		IF SIf.Par.bolEnableDoublePaperDetection THEN
			me.StateMachine.intStateNext := Base_PLC.cSTA_ERROR;
		END_IF
	ELSE	
		CASE me.SubStateMachine.intState OF
			// substate Wait paper - wait for the next paper if the buffer was empty
			// ------------------------------------------------------------------------
			PBC_CmdState.cSUB_WAITPAPER:
				IF NOT SIf.In.bolPaperAvailableExit.intern THEN
					IF SIf.In.bolCapacityReached.intern OR SIf.In.bolPaperAvailableEntry.intern THEN
						me.SubStateMachine.intStateNext := PBC_CmdState.cSUB_POSITIONSTARTbusy;
					END_IF
				ELSE
					me.SubStateMachine.intStateNext := cSUB_EVALUATEEJECT;
				END_IF
				
			// substate PositionStart busy
			// ------------------------------------------------------------------------
			PBC_CmdState.cSUB_POSITIONSTARTbusy:
				IF NOT SIf.In.bolPaperAvailableExit.intern THEN
					SIf.Cur.bolPaperBeforeEjectAvailable := SIf.In.bolCapacityReached.intern OR SIf.In.bolPaperAvailableEntry.intern;
					pDeStackerCIf^.Job.intACmd := BASE_PLC.cCMD_RUN;
					me.SubStateMachine.intStateNext := PBC_CmdState.cSUB_POSITIONbusy;
				ELSE
					me.SubStateMachine.intStateNext := cSUB_EVALUATEEJECT;
				END_IF
	
			// substate Position busy
			// ------------------------------------------------------------------------
			PBC_CmdState.cSUB_POSITIONbusy:
				IF me.SubStateMachine.udiTimeInState_ms <= SIf.Par.udiPaperTransportTime THEN
					IF SIf.In.bolPaperAvailableExit.intern THEN
						m_intRetry := 0;
						pDeStackerCIf^.Job.intACmd := BASE_PLC.cCMD_STOP;
						me.SubStateMachine.intStateNext := PBC_CmdState.cSUB_POSITIONSTOPbusy;
					END_IF
				ELSE
					IF SIf.Cur.bolPaperBeforeEjectAvailable OR SIf.In.bolCapacityReached.intern OR SIf.In.bolPaperAvailableEntry.intern THEN
						IF DINT_TO_UDINT(m_intRetry) < SIf.Par.udiPaperInjectRetries THEN
							pDeStackerCIf^.Job.intACmd := BASE_PLC.cCMD_STOP;
							m_intRetry := m_intRetry + 1;
							pfbAlarmCtrl^.setAlarm(CIf.Info.intCtrlId,INT_TO_UINT(E_ALM_PBC.PaperInjectRetry),m_intRetry,ADR(SIf.Alm),E_AlmState.RST,CIf.Job.eMe_ActivAlmClass);
							me.SubStateMachine.intStateNext := PBC_CmdState.cSUB_POSITIONRETRYSTOP;	
						ELSE
							m_intRetry := 0;
							pfbAlarmCtrl^.setAlarm(CIf.Info.intCtrlId,INT_TO_UINT(E_ALM_PBC.PaperInject),0,ADR(SIf.Alm),E_AlmState.RST,CIf.Job.eMe_ActivAlmClass);
							me.StateMachine.intStateNext := Base_PLC.cSTA_ERROR;	
						END_IF
					ELSE
						m_intRetry := 0;
						pDeStackerCIf^.Job.intACmd := BASE_PLC.cCMD_STOP;
						me.SubStateMachine.intStateNext := PBC_CmdState.cSUB_POSITIONSTOPbusy;
					END_IF 
				END_IF

				// Simulation
				IF CIf.SwCfg.bolSimulation THEN
					IF (me.SubStateMachine.udiTimeInState_ms > SIf.Par.udiSimPaperTransportTime) AND NOT SIf.In.bolPaperAvailableExit.intern THEN
						SIf.In.bolPaperAvailableExit.intern := TRUE;	
					END_IF
				END_IF
				// -----------------------------------
	
			// Wait that the moto stops
			// ------------------------------------------------------------------------
			PBC_CmdState.cSUB_POSITIONRETRYSTOP:
				IF pDeStackerCIf^.Job.intState = BASE_PLC.cSTA_STOP THEN
					me.SubStateMachine.intStateNext := PBC_CmdState.cSUB_POSITIONRETRYDELAY;
				END_IF

			// Stop the motor and way for x ms
			// ------------------------------------------------------------------------
			PBC_CmdState.cSUB_POSITIONRETRYDELAY:
				IF me.SubStateMachine.udiTimeInState_ms > SIf.Par.udiPaperInjectRetryPauseTime_ms THEN
					me.SubStateMachine.intStateNext := PBC_CmdState.cSUB_POSITIONSTARTbusy;
				END_IF

			// substate PositionStop busy
			// ------------------------------------------------------------------------
			PBC_CmdState.cSUB_POSITIONSTOPbusy:
				IF pDeStackerCIf^.Job.intState = BASE_PLC.cSTA_STOP THEN
					me.SubStateMachine.intStateNext := PBC_CmdState.cSUB_EVALUATEEJECT;
				END_IF

			// substate Evaluate Eject
			// ------------------------------------------------------------------------
			PBC_CmdState.cSUB_EVALUATEEJECT:
				bolSaberStopDestack		:= SIf.Par.bolStopReleaseItems AND SIf.Cfg.bolEnableSaberStopDeStack;

				// Eject next paper if there are still paper to edject or endless ejection
				IF (((SIf.Cur.uinPaperToEjectCount > 0) AND NOT SIf.Par.bolAutomaticMode AND NOT bolSaberStopDestack) 
					OR (SIf.Par.bolAutomaticMode AND NOT bolSaberStopDestack)) THEN 
					// Make a delay from sheet to sheet if it is not the first sheet
					IF SIf.In.bolPaperAvailableExit.intern THEN
						IF   (SIf.Cur.uinSheetToSheetTime > SIf.Par.udiSheetToSheetTime) 
						  OR ((SIf.Cur.uinPaperToEjectCount = SIf.Cur.uinPaperToEjectParameter) AND NOT SIf.Par.bolAutomaticMode) THEN
							SIf.Cur.uinSheetToSheetTime := 0;
							me.SubStateMachine.intStateNext := PBC_CmdState.cSUB_EJECTSTARTbusy;
						END_IF
					ELSE
						me.SubStateMachine.intStateNext := PBC_CmdState.cSUB_WAITPAPER;
					END_IF
				ELSE
					me.StateMachine.intStateNext := cSTA_STOPBusy;
				END_IF
	
			// substate EjectStart busy
			// ------------------------------------------------------------------------
			PBC_CmdState.cSUB_EJECTSTARTbusy:
				pDeStackerCIf^.Job.intACmd := BASE_PLC.cCMD_RUN;
				SIf.Cur.uinPaperToPaperTime_ms := UDINT_TO_UINT((m_uinPaperHight_mm + 100) * 1000 / p_fbDeStacker^.CtrlSIf^.Par.rBeltParam.uinBeltSpeed);
				SIf.Par.udiSimPaperToPaperTransportTime := SIf.Cur.uinPaperToPaperTime_ms / 3; 
				me.SubStateMachine.intStateNext := PBC_CmdState.cSUB_EJECTbusy;
	
			// substate Eject busy
			// ------------------------------------------------------------------------
			PBC_CmdState.cSUB_EJECTbusy:
				IF NOT SIf.In.bolPaperAvailableExit.intern AND NOT SIf.Cfg.bolUseTurnTableSensorForEject THEN
					pDeStackerCIf^.Job.intACmd := BASE_PLC.cCMD_STOP;
					me.SubStateMachine.intStateNext := PBC_CmdState.cSUB_EJECTSTOPbusy;
				END_IF
	
				IF SIf.In.bolTurnTableMiddleSensor.intern AND SIf.Cfg.bolUseTurnTableSensorForEject THEN
					pDeStackerCIf^.Job.intACmd := BASE_PLC.cCMD_STOP;
					me.SubStateMachine.intStateNext := PBC_CmdState.cSUB_WAITPAPERGONETABLE;
				END_IF
				
				IF (me.SubStateMachine.udiTimeInState_ms > SIf.Cur.uinPaperToPaperTime_ms) THEN
					pfbAlarmCtrl^.setAlarm(CIf.Info.intCtrlId,INT_TO_UINT(E_ALM_PBC.PaperTransport),0,ADR(SIf.Alm),E_AlmState.RST,CIf.Job.eMe_ActivAlmClass);
					me.StateMachine.intStateNext := Base_PLC.cSTA_ERROR;	
				END_IF

				// Simulation
				IF CIf.SwCfg.bolSimulation THEN
					IF (me.SubStateMachine.udiTimeInState_ms > SIf.Par.udiSimPaperToPaperTransportTime) THEN
						IF SIf.Cfg.bolUseTurnTableSensorForEject THEN
							SIf.In.bolTurnTableMiddleSensor.intern := TRUE;
						ELSE
							SIf.In.bolPaperAvailableExit.intern := FALSE;	
						END_IF	
					END_IF
				END_IF
				// -----------------------------------
	
			// substate Wait Paper Gone Table - Wait until the paper is gone from the turn table
			// ------------------------------------------------------------------------
			PBC_CmdState.cSUB_WAITPAPERGONETABLE:
				IF NOT SIf.In.bolTurnTableMiddleSensor.intern THEN
					me.SubStateMachine.intStateNext := PBC_CmdState.cSUB_EJECTSTOPbusy;
				END_IF

				// Simulation
				IF CIf.SwCfg.bolSimulation THEN
					IF (me.SubStateMachine.udiTimeInState_ms > SIf.Par.udiSimPaperToPaperTransportTime) THEN
						SIf.In.bolTurnTableMiddleSensor.intern := FALSE;
					END_IF
				END_IF
				// -----------------------------------

	
			// substate EjectStop busy
			// ------------------------------------------------------------------------
			PBC_CmdState.cSUB_EJECTSTOPbusy:
				IF pDeStackerCIf^.Job.intState = BASE_PLC.cSTA_STOP THEN
					IF SIf.Cur.uinPaperToEjectCount > 0 THEN
						SIf.Cur.uinPaperToEjectCount := SIf.Cur.uinPaperToEjectCount - 1;
					END_IF
	
					me.SubStateMachine.intStateNext := PBC_CmdState.cSUB_POSITIONSTARTbusy;
				END_IF
		END_CASE
	END_IF
	
	CASE me.SubStateMachine.intState OF
		PBC_CmdState.cSUB_WAITPAPER,
		PBC_CmdState.cSUB_EVALUATEEJECT:
			IF (me.intCmd = BASE_PLC.cCMD_STOP) THEN 
					me.StateMachine.intStateNext := BASE_PLC.cSTA_STOPBusy;
			END_IF
	END_CASE
	
	SIf.Cur.uinSheetToSheetTime := UDINT_TO_UINT(SIf.Cur.uinSheetToSheetTime + me.FUBInfo.udiSample_ms);
END_IF


//--------------------------------------------------------------------------------------
// Exit action
IF (me.StateMachine.intState<>me.StateMachine.intStateNext) THEN
	me.SubStateMachine.intState 	:= BASE_PLC.cSTA_INITIALIZED;
	me.SubStateMachine.intStateNext := BASE_PLC.cSTA_INITIALIZED;
END_IF
END_METHOD

{attribute 'object_name' := 'sta_RUNbusy'}
METHOD PROTECTED sta_RUNbusy : BOOL
// state implemetation
//--------------------------------------------------------------------------------------
// Entry action
IF (me.StateMachine.intState<>me.StateMachine.intStateLastCycle) THEN
	me.StateMachine.intStateLastCycle := me.StateMachine.intState;

	IF (CIf.SwCfg.bolSimulation) THEN
		SIf.In.bolCapacityReached.intern := FALSE;
		SIf.In.bolPaperAvailableEntry.intern := TRUE;
		SIf.In.bolPaperAvailableExit.intern := TRUE;
	END_IF

	SIf.Out.bolAirOn.intern := TRUE;
	
	pDeStackerCIf^.Job.intACmd := BASE_PLC.cCMD_STOP;
	pBeltCIf^.Job.intACmd := BASE_PLC.cCMD_RUN;
	
	// clear alarm
	pfbAlarmCtrl^.setAlarm(CIf.Info.intCtrlId,INT_TO_UINT(E_ALM_PBC.DoNotReleaseItems),0,ADR(SIf.Alm),E_AlmState.CLR,CIf.Job.eMe_ActivAlmClass);
END_IF


//--------------------------------------------------------------------------------------
// Cyclic action
IF (me.StateMachine.intState=me.StateMachine.intStateLastCycle) THEN
	IF SIf.Par.bolAutomaticMode THEN
		SIf.Cur.uinPaperToEjectParameter := 0;
		SIf.Cur.uinPaperToEjectCount := 0;
		me.StateMachine.intStateNext := BASE_PLC.cSTA_RUN;
	ELSE	
		IF me.intCmd = PBC_CmdState.cCMD_SINGLE THEN
			SIf.Cur.uinPaperToEjectParameter := 1;
			SIf.Cur.uinPaperToEjectCount := 1;
	
			IF NOT SIf.In.bolPaperAvailableExit.intern AND NOT SIf.In.bolPaperAvailableEntry.intern THEN
				pfbAlarmCtrl^.setAlarm(CIf.Info.intCtrlId,INT_TO_UINT(E_ALM_PBC.BufferEmpty),0,ADR(SIf.Alm),E_AlmState.RST,CIf.Job.eMe_ActivAlmClass);
			END_IF
	
			me.StateMachine.intStateNext := BASE_PLC.cSTA_RUN;
		ELSE
			IF me.StateMachine.intStateHistory = Base_PLC.cSTA_OFF THEN
				CIf.Job.intACmd := cCMD_DONE;
				CIf.Job.intMCmd := cCMD_DONE;
				me.StateMachine.intStateNext := BASE_PLC.cSTA_STOPBusy;
			ELSE
				SIf.Cur.uinPaperToEjectParameter := UDINT_TO_UINT(SIf.Par.udiSheetToEject);
				SIf.Cur.uinPaperToEjectCount := UDINT_TO_UINT(SIf.Par.udiSheetToEject);
		
				IF SIf.Par.udiSheetToEject > 0 THEN
					me.StateMachine.intStateNext := BASE_PLC.cSTA_RUN;
				ELSE
					CIf.Job.intACmd := cCMD_DONE;
					CIf.Job.intMCmd := cCMD_DONE;
					me.StateMachine.intStateNext := BASE_PLC.cSTA_STOPBusy;
				END_IF
			END_IF
		END_IF
	END_IF
END_IF


//--------------------------------------------------------------------------------------
// Exit action
IF (me.StateMachine.intState<>me.StateMachine.intStateNext) THEN
	;
END_IF
END_METHOD

{attribute 'object_name' := 'sta_STOP'}
METHOD PROTECTED sta_STOP : BOOL
// state implemetation
//--------------------------------------------------------------------------------------
// Entry action
IF (me.StateMachine.intState<>me.StateMachine.intStateLastCycle) THEN
	me.StateMachine.intStateLastCycle := me.StateMachine.intState;

	IF CIf.SwCfg.bolSimulation THEN
		SIf.In.bolPaperAvailableEntry.intern := TRUE;
		SIf.In.bolDoublePaperDetection.intern := FALSE;	
		SIf.In.bolPaperAvailableExit.intern := FALSE;	
		SIf.In.bolCapacityReached.intern := TRUE;
	END_IF
	
	IF me.intCmd = Base_PLC.cCMD_RUN THEN
		CIf.Job.intACmd := Base_PLC.cCMD_DONE;
		CIf.Job.intMCmd := Base_PLC.cCMD_DONE;
	END_IF
	
	me.SubStateMachine.intState 	:= PBC_CmdState.cSUB_POSITIONSTARTbusy;
	me.SubStateMachine.intStateNext := PBC_CmdState.cSUB_POSITIONSTARTbusy;
END_IF

//--------------------------------------------------------------------------------------
// Cyclic action
IF (me.StateMachine.intState=me.StateMachine.intStateLastCycle) THEN
	CASE me.SubStateMachine.intState OF
		// substate Wait paper - wait for the next paper if the buffer was empty
		// ------------------------------------------------------------------------
		PBC_CmdState.cSUB_WAITPAPER:
			IF SIf.In.bolPaperAvailableExit.intern THEN
				me.SubStateMachine.intStateNext := PBC_CmdState.cSUB_READYEJECT;
			ELSE
				IF SIf.In.bolCapacityReached.intern OR SIf.In.bolPaperAvailableEntry.intern THEN
					me.SubStateMachine.intStateNext := PBC_CmdState.cSUB_POSITIONSTARTbusy;
				END_IF
			END_IF
			
		// substate Wait paper - wait for the next paper if the buffer was empty
		// ------------------------------------------------------------------------
		PBC_CmdState.cSUB_POSITIONSTARTbusy:
			IF NOT SIf.In.bolPaperAvailableExit.intern THEN
				SIf.Cur.bolPaperBeforeEjectAvailable := SIf.In.bolCapacityReached.intern OR SIf.In.bolPaperAvailableEntry.intern;
				pDeStackerCIf^.Job.intACmd := BASE_PLC.cCMD_RUN;
				me.SubStateMachine.intStateNext := PBC_CmdState.cSUB_POSITIONbusy;
			ELSE
				me.SubStateMachine.intStateNext := cSUB_READYEJECT;
			END_IF

		// substate Wait paper - wait for the next paper if the buffer was empty
		// ------------------------------------------------------------------------
		PBC_CmdState.cSUB_POSITIONbusy:
			IF me.SubStateMachine.udiTimeInState_ms > SIf.Par.udiPaperTransportTime THEN
				IF SIf.Cur.bolPaperBeforeEjectAvailable OR SIf.In.bolCapacityReached.intern OR SIf.In.bolPaperAvailableEntry.intern THEN
					pfbAlarmCtrl^.setAlarm(CIf.Info.intCtrlId,INT_TO_UINT(E_ALM_PBC.PaperTransport),0,ADR(SIf.Alm),E_AlmState.RST,CIf.Job.eMe_ActivAlmClass);
					me.StateMachine.intStateNext := Base_PLC.cSTA_ERROR;	
				ELSE
					pDeStackerCIf^.Job.intACmd := BASE_PLC.cCMD_STOP;
					me.SubStateMachine.intStateNext := PBC_CmdState.cSUB_POSITIONSTOPbusy;
				END_IF 
			ELSE
				IF SIf.In.bolPaperAvailableExit.intern THEN
					pDeStackerCIf^.Job.intACmd := BASE_PLC.cCMD_STOP;
					me.SubStateMachine.intStateNext := PBC_CmdState.cSUB_POSITIONSTOPbusy;
				END_IF
			END_IF
			
			// Simulation
			IF CIf.SwCfg.bolSimulation THEN
				IF (me.SubStateMachine.udiTimeInState_ms > SIf.Par.udiSimPaperTransportTime) AND NOT SIf.In.bolPaperAvailableExit.intern THEN
					SIf.In.bolPaperAvailableExit.intern := TRUE;	
				END_IF
			END_IF
			// -----------------------------------

		// substate Wait paper - wait for the next paper if the buffer was empty
		// ------------------------------------------------------------------------
		PBC_CmdState.cSUB_POSITIONSTOPbusy:
			IF pDeStackerCIf^.Job.intState = BASE_PLC.cSTA_STOP THEN
				IF SIf.In.bolPaperAvailableExit.intern THEN
					me.SubStateMachine.intStateNext := PBC_CmdState.cSUB_READYEJECT;
				ELSE
					me.SubStateMachine.intStateNext := PBC_CmdState.cSUB_WAITPAPER;
				END_IF
			END_IF
		PBC_CmdState.cSUB_READYEJECT:
			IF NOT SIf.In.bolPaperAvailableExit.intern THEN
				me.SubStateMachine.intStateNext := PBC_CmdState.cSUB_WAITPAPER;
			END_IF
	END_CASE

	CASE me.SubStateMachine.intState OF
		PBC_CmdState.cSUB_WAITPAPER,
		PBC_CmdState.cSUB_READYEJECT:
			IF me.intCmd = PBC_CmdState.cCMD_SINGLE THEN
				me.StateMachine.intStateNext := BASE_PLC.cSTA_RUNBusy;
			END_IF
		
			IF ((me.intCmd = BASE_PLC.cCMD_RUN) AND (NOT SIf.Par.bolStopReleaseItems AND SIf.Cfg.bolEnableSaberStopDeStack))
				OR ((me.intCmd = BASE_PLC.cCMD_RUN) AND NOT SIf.Cfg.bolEnableSaberStopDeStack) THEN
				me.StateMachine.intStateNext := BASE_PLC.cSTA_RUNBusy;
			END_IF

			IF (SIf.Par.bolAutomaticMode AND (NOT SIf.Par.bolStopReleaseItems AND SIf.Cfg.bolEnableSaberStopDeStack))
				OR (SIf.Par.bolAutomaticMode AND NOT SIf.Cfg.bolEnableSaberStopDeStack) THEN
				me.StateMachine.intStateNext := BASE_PLC.cSTA_RUNBusy;
			END_IF
	END_CASE
END_IF


//--------------------------------------------------------------------------------------
// Exit action
IF (me.StateMachine.intState<>me.StateMachine.intStateNext) THEN
	me.SubStateMachine.intState 	:= BASE_PLC.cSTA_INITIALIZED;
	me.SubStateMachine.intStateNext := BASE_PLC.cSTA_INITIALIZED;
END_IF
END_METHOD

{attribute 'object_name' := 'sta_STOPbusy'}
METHOD PROTECTED sta_STOPbusy : BOOL
// state implemetation
//--------------------------------------------------------------------------------------
// Entry action
IF (me.StateMachine.intState<>me.StateMachine.intStateLastCycle) THEN
	me.StateMachine.intStateLastCycle := me.StateMachine.intState;

	pDeStackerCIf^.Job.intACmd := BASE_PLC.cCMD_STOP;
	
	// set alarm
	pfbAlarmCtrl^.setAlarm(CIf.Info.intCtrlId,INT_TO_UINT(E_ALM_PBC.DoNotReleaseItems),0,ADR(SIf.Alm),E_AlmState.SET,CIf.Job.eMe_ActivAlmClass);
END_IF


//--------------------------------------------------------------------------------------
// Cyclic action
IF (me.StateMachine.intState=me.StateMachine.intStateLastCycle) THEN
	me.StateMachine.intStateNext := BASE_PLC.cSTA_STOP;
END_IF


//--------------------------------------------------------------------------------------
// Exit action
IF (me.StateMachine.intState<>me.StateMachine.intStateNext) THEN
	;
END_IF
END_METHOD

{attribute 'object_name' := 'StateMachine'}
METHOD PROTECTED StateMachine : BOOL
SUPER^.StateMachine();

// main statemachine of base controller
CASE me.StateMachine.intState OF
	BASE_PLC.cSTA_RUN:
		THIS^.sta_RUN();
	BASE_PLC.cSTA_RUNBusy:
		THIS^.sta_RUNbusy();
    BASE_PLC.cSTA_STOPBusy: 
        THIS^.sta_STOPbusy();
    BASE_PLC.cSTA_STOP: 
        THIS^.sta_STOP();
	PBC_CmdState.cSTA_INITbusy:
		THIS^.sta_INITbusy();
END_CASE;
END_METHOD

END_FUNCTION_BLOCK

// POUs/Controller/Lvl2/PCE [Paper Belt Corner Element]/helper/cycle_Pce
FUNCTION cycle_Pce : BOOL
VAR_INPUT
	pPce: POINTER TO T_PCE;
END_VAR

pPce^.ctrl.fbPce_PtbIn_Umc.In_bolEmoOk				:= pPce^.io.In_bolUmcIn_EmoOk;
pPce^.ctrl.fbPce_PtbIn_Umc.In_uinStatus				:= pPce^.io.In_uinUmcIn_Status;
pPce^.ctrl.fbPce_PtbIn_Umc.In_intMotorActualSpeed	:= pPce^.io.In_uinUmcIn_ActualSpeed;
pPce^.ctrl.fbPce_PtbIn_Umc.In_uinMotorSetSpeed		:= pPce^.io.In_uinUmcIn_SetSpeed;
pPce^.ctrl.fbPce_PtbIn_Umc.In_uinECATState			:= pPce^.io.In_uinUmcIn_ECatState;
pPce^.ctrl.fbPce_PtbIn_Umc.In_strNetId				:= pPce^.io.In_strUmcIn_ECatNetId;
pPce^.ctrl.fbPce_PtbIn_Umc.In_uintPort				:= pPce^.io.In_uinUmcIn_ECatPort;
pPce^.ctrl.fbPce_PtbIn_Umc();
pPce^.io.Out_uinUmcIn_SetSpeed						:= pPce^.ctrl.fbPce_PtbIn_Umc.Out_uinSpeedSetpoint;
pPce^.io.Out_uinUmcIn_Control						:= pPce^.ctrl.fbPce_PtbIn_Umc.Out_uinControl;

pPce^.ctrl.fbPce_PtbIn_Vpc.In_bolPumpOk				:= pPce^.io.In_bolVpc_PumpOk;
pPce^.ctrl.fbPce_PtbIn_Vpc.In_bolVacuumOk			:= pPce^.io.In_bolVpc_VacuumSensor;
pPce^.ctrl.fbPce_PtbIn_Vpc();
pPce^.io.Out_bolVpc_PumpOn							:= pPce^.ctrl.fbPce_PtbIn_Vpc.Out_bolVaccumPumpOn;

pPce^.ctrl.fbPce_PtbIn.In_bolBeltEntrySensor		:= pPce^.io.In_bolInputSensor;
pPce^.ctrl.fbPce_PtbIn.In_bolBeltExitSensor			:= pPce^.io.In_bolCornerSensor;
pPce^.ctrl.fbPce_PtbIn();

pPce^.ctrl.fbPce_PtbOut_Umc.In_bolEmoOk				:= pPce^.io.In_bolUmcIn_EmoOk;
pPce^.ctrl.fbPce_PtbOut_Umc.In_uinStatus			:= pPce^.io.In_uinUmcOut_Status;
pPce^.ctrl.fbPce_PtbOut_Umc.In_intMotorActualSpeed	:= pPce^.io.In_uinUmcOut_ActualSpeed;
pPce^.ctrl.fbPce_PtbOut_Umc.In_uinMotorSetSpeed		:= pPce^.io.In_uinUmcOut_SetSpeed;
pPce^.ctrl.fbPce_PtbOut_Umc.In_uinECATState			:= pPce^.io.In_uinUmcOut_ECatState;
pPce^.ctrl.fbPce_PtbOut_Umc.In_strNetId				:= pPce^.io.In_strUmcOut_ECatNetId;
pPce^.ctrl.fbPce_PtbOut_Umc.In_uintPort				:= pPce^.io.In_uinUmcOut_ECatPort;
pPce^.ctrl.fbPce_PtbOut_Umc();
pPce^.io.Out_uinUmcOut_SetSpeed						:= pPce^.ctrl.fbPce_PtbOut_Umc.Out_uinSpeedSetpoint;
pPce^.io.Out_uinUmcOut_Control						:= pPce^.ctrl.fbPce_PtbOut_Umc.Out_uinControl;

pPce^.ctrl.fbPce_PtbOut.In_bolBeltEntrySensor		:= pPce^.io.In_bolCornerSensor;
pPce^.ctrl.fbPce_PtbOut.In_bolBeltExitSensor		:= pPce^.io.In_bolOutputSensor;
pPce^.ctrl.fbPce_PtbOut();

pPce^.ctrl.fbPce.In_bolPaperAvailable				:=pPce^.io.In_bolCornerSensor;
pPce^.ctrl.fbPce();
pPce^.io.Out_bolVacuumValveIn						:= pPce^.ctrl.fbPce.Out_bolVacuumValveIn;
pPce^.io.Out_bolVacuumValveOut						:= pPce^.ctrl.fbPce.Out_bolVacuumValveOut;

END_FUNCTION

// POUs/Controller/Lvl2/PCE [Paper Belt Corner Element]/helper/init_Pce
FUNCTION init_Pce : BOOL
VAR_INPUT
	pPce			: POINTER TO T_PCE;
	/// instance array of all controller instances
	pCtrlInst		: POINTER TO fb_CtrlBase;
	/// common interface array of all controllers (main use for PLC)
	pCtrlCIf		: POINTER TO T_Ctrl_CIf;
END_VAR

pPce^.ctrl.fbPce_PtbIn_Vpc.iniAllCtrlArrays(pCtrlInst,pCtrlCIf,pPce^.id.Pce_PtbIn_Vpc);
pPce^.ctrl.fbPce_PtbIn_Umc.iniAllCtrlArrays(pCtrlInst,pCtrlCIf,pPce^.id.Pce_PtbIn_Umc);
pPce^.ctrl.fbPce_PtbIn.iniAllCtrlArrays(pCtrlInst,pCtrlCIf,pPce^.id.Pce_PtbIn);
pPce^.ctrl.fbPce_PtbIn.Drive := ADR(pPce^.ctrl.fbPce_PtbIn_Umc);
pPce^.ctrl.fbPce_PtbIn.VacuumPump := ADR(pPce^.ctrl.fbPce_PtbIn_Vpc);

pPce^.ctrl.fbPce_PtbOut_Umc.iniAllCtrlArrays(pCtrlInst,pCtrlCIf,pPce^.id.Pce_PtbOut_Umc);
pPce^.ctrl.fbPce_PtbOut.iniAllCtrlArrays(pCtrlInst,pCtrlCIf,pPce^.id.Pce_PtbOut);
pPce^.ctrl.fbPce_PtbOut.Drive := ADR(pPce^.ctrl.fbPce_PtbOut_Umc);

pPce^.ctrl.fbPce.iniAllCtrlArrays(pCtrlInst,pCtrlCIf,pPce^.id.Pce);
pPce^.ctrl.fbPce.DriveIn := ADR(pPce^.ctrl.fbPce_PtbIn);
pPce^.ctrl.fbPce.DriveOut := ADR(pPce^.ctrl.fbPce_PtbOut);

END_FUNCTION

// POUs/Controller/Lvl2/PCE [Paper Belt Corner Element]/FB_PCE
FUNCTION_BLOCK FB_PCE EXTENDS FB_CtrlBase
VAR_INPUT
	In_bolPaperAvailable: BOOL;
END_VAR
VAR_OUTPUT
	Out_bolVacuumValveIn: BOOL;
	Out_bolVacuumValveOut: BOOL;
END_VAR
VAR
	/// Specific interface struct for public access
	SIf: T_Ctrl_SIf_PCE;
	///pointer to function block
	p_fbMotorIn: POINTER TO FB_PTB;
	pMotorInCIf: POINTER TO T_Ctrl_CIf;
	p_fbMotorOut: POINTER TO FB_PTB;
	pMotorOutCIf: POINTER TO T_Ctrl_CIf;
END_VAR

(*__________________________________________________________________________________________________
¦	
¦	Vistaprint Schweiz GmbH
¦	CH - 8401 Winterthur
¦
¦	www.vistaprint.ch - info@vistaprint.ch
¦___________________________________________________________________________________________________

Function desription:
Vacuum Pump implementation. 


History:
Version		Date			Author		Comment
---------------------------------------------------------------------------------------------------
0.00.1		09.07.2013		PC			Start history
___________________________________________________________________________________________________*)


SUPER^();

{attribute 'object_name' := 'Always'}
METHOD PROTECTED Always : BOOL
SUPER^.Always();

// ----------------------------------------------------------------------------------
// cyclic actions outside of statemachine
IF (me.StateMachine.intState<>cSTA_SINGLE_ANSWER) THEN
	
	; // always error supervision
	
END_IF

// ----------------------------------------------------------------------------------
// Conditions Always
IF (((me.Alarm.eActivAlmClass=E_AlmClass.EOFF) OR (me.Alarm.eActivAlmClass=E_AlmClass.OFF) OR (me.intCmd=cCMD_OFF) OR (me.intCmd=BASE_PLC.cCMD_EOFF))
		 AND (me.StateMachine.intState<>cSTA_ERROR) AND (me.StateMachine.intState<>cSTA_ERRORQuit) AND
		(me.StateMachine.intState<>cSTA_OFF) AND (me.StateMachine.intState<>cSTA_OFFBusy)) THEN
	// alarm evt EOFF, OFF or cmd off
	me.StateMachine.intStateNext := cSTA_OFFBusy;
END_IF
END_METHOD

{attribute 'object_name' := 'CtrlInit'}
METHOD CtrlInit : BOOL
SUPER^.CtrlInit();

pMotorInCIf := p_fbMotorIn^.CtrlCIf;
pMotorOutCIf := p_fbMotorOut^.CtrlCIf;

AddChild(p_fbMotorIn^);
AddChild(p_fbMotorOut^);
END_METHOD

PROPERTY PUBLIC CtrlSIf : POINTER TO T_Ctrl_SIf_PCE
GET
CtrlSIf := ADR(SIf);
END_GET
END_PROPERTY

PROPERTY DriveIn : POINTER TO FB_PTB
GET
DriveIn := p_fbMotorIn;
END_GET
SET
p_fbMotorIn := DriveIn;
END_SET
END_PROPERTY

PROPERTY DriveOut : POINTER TO FB_PTB
GET
DriveOut := p_fbMotorOut;
END_GET
SET
p_fbMotorOut := DriveOut;
END_SET
END_PROPERTY

{attribute 'object_name' := 'FB_init'}
METHOD FB_init : BOOL
VAR_INPUT
	/// if TRUE, the retain variables are initialized (warm start / cold start)
	bInitRetains: BOOL;
	/// if TRUE, the instance afterwards gets moved into the copy code (online change)
	bInCopyCode: BOOL;
END_VAR
VAR
	iIdx: UINT;
	iLength: UINT;
END_VAR
//------------------------------------------------------------------------------------------------------------------------
// to manually change in new FUB implementation!!!
// define valid commands for this controller
iLength := SIZEOF(CIf.Job.aCmdList)/SIZEOF(CIf.Job.aCmdList[0]);
iIdx := 0;

WHILE (iIdx < iLength) AND (CIf.Job.aCmdList[iIdx].intCmd <> cCMD_INITIALIZED) DO
	iIdx := iIdx + 1; 
END_WHILE

IF (iIdx < iLength) THEN
// Add configuration of own comands	
	CIf.Job.aCmdList[iIdx].intCmd := BASE_PLC.cCMD_RUN;
	CIf.Job.aCmdList[iIdx].strName := 'Run'; 
	CIf.Job.aCmdList[iIdx].bolAvailable := TRUE;
	iIdx := iIdx + 1;
	CIf.Job.aCmdList[iIdx].intCmd := BASE_PLC.cCMD_STOP;
	CIf.Job.aCmdList[iIdx].strName := 'Stop'; 
	CIf.Job.aCmdList[iIdx].bolAvailable := TRUE;
ELSE
	// Error if the aCmdList Array is to small
END_IF

// set name of class/typ
CIf.Info.strType := 'FB_PCE';
CIf.Info.strFullName := 'Paper Corner Element';

// set alarm class

SIf.Alm[E_ALM_PCE.PaperSensorError].eAlmClass := Base_PLC.E_AlmClass.TSTOP;
SIf.Alm[E_ALM_PCE.PaperSensorError].strText := 'Paper detected to long' ;


//*******************************************************************************
// initial values
//*******************************************************************************

// software configuration
CIf.SwCfg.bolExist := TRUE;
CIf.SwCfg.bolEnable := TRUE;
CIf.SwCfg.bolSimulation := FALSE;

// parameter
SIf.Par.uinPaperExitTime_ms			:= 3000;
SIf.Par.uinSimPaperExitTime_ms		:= SIf.Par.uinPaperExitTime_ms / 2;
SIf.Par.uinPaperEntryDelayTime_ms   := 220;
END_METHOD

{attribute 'object_name' := 'getCmdState'}
METHOD PROTECTED getCmdState : STRING
VAR_INPUT
	intCmdState: INT;
	bolState: BOOL;
END_VAR
getCmdState := SUPER^.getCmdState(intCmdState:=intCmdState,bolState:=bolState); // get global/base defined cmds/states
END_METHOD

{attribute 'object_name' := 'getCtrlSIf'}
METHOD getCtrlSIf : POINTER TO T_Ctrl_SIf_PCE
getCtrlSIf := ADR(SIf);
END_METHOD

{attribute 'object_name' := 'IoInBridge'}
METHOD PROTECTED IoInBridge : BOOL
// digitale and analoge inputs read from hardware or forcing
SIf.In.bolPaperAvailable.map := THIS^.In_bolPaperAvailable;

IF (CIf.SwCfg.bolSimulation = FALSE) THEN
	getInBol(CIf.Job.bolIoForce,ADR(SIf.In.bolPaperAvailable));
ELSE
	;//simulation of global IO
END_IF
END_METHOD

{attribute 'object_name' := 'IoOutBridge'}
METHOD PROTECTED IoOutBridge : BOOL
VAR
	bolSwitchValvesOff: BOOL;
END_VAR
// digitale and analoge inputs read from hardware or forcing
IF (CIf.SwCfg.bolSimulation = FALSE) THEN
	setOutBol(CIf.Job.bolIoForce ,ADR(SIf.Out.bolVacuumValveIn));
	setOutBol(CIf.Job.bolIoForce ,ADR(SIf.Out.bolVacuumValveOut));

	THIS^.Out_bolVacuumValveIn := SIf.Out.bolVacuumValveIn.map;
	THIS^.Out_bolVacuumValveOut := SIf.Out.bolVacuumValveOut.map;
END_IF
END_METHOD

ACTION PaperExitValveActive:
SIf.Out.bolVacuumValveIn.intern := FALSE;
SIf.Out.bolVacuumValveOut.intern := TRUE;
END_ACTION

ACTION PaperInputValveActive:
SIf.Out.bolVacuumValveIn.intern := TRUE;
SIf.Out.bolVacuumValveOut.intern := FALSE;
END_ACTION

{attribute 'object_name' := 'sta_ERROR'}
METHOD PROTECTED sta_ERROR : BOOL
// state implemetation
//--------------------------------------------------------------------------------------
// Entry action
	IF (me.StateMachine.intState<>me.StateMachine.intStateLastCycle) THEN
		me.StateMachine.intStateHistory := me.StateMachine.intStateLastCycle; // -> possibillity to go back to state before error
		me.StateMachine.intStateLastCycle := me.StateMachine.intState;
		p_fbMotorIn^.CtrlCIf^.Job.intACmd := BASE_PLC.cCMD_STOP;
		p_fbMotorOut^.CtrlCIf^.Job.intACmd := BASE_PLC.cCMD_STOP;
	END_IF


//--------------------------------------------------------------------------------------
// Cyclic action
	IF (me.StateMachine.intState=me.StateMachine.intStateLastCycle) THEN
		
		;
		
		
		// State Change Condition
		IF (CIf.Job.bolAlmReset = TRUE) THEN
			me.StateMachine.intStateNext := cSTA_ERRORQuit;
		END_IF
	END_IF




//--------------------------------------------------------------------------------------
// Exit action
	IF (me.StateMachine.intState<>me.StateMachine.intStateNext) THEN
		;
	END_IF
END_METHOD

{attribute 'object_name' := 'sta_ERRORQuit'}
METHOD PROTECTED sta_ERRORQuit : BOOL
// state implemetation
//--------------------------------------------------------------------------------------
// Entry action
	IF (me.StateMachine.intState<>me.StateMachine.intStateLastCycle) THEN
		me.StateMachine.intStateLastCycle := me.StateMachine.intState;
		
	END_IF


//--------------------------------------------------------------------------------------
// Cyclic action
	IF (me.StateMachine.intState=me.StateMachine.intStateLastCycle) THEN
		
		;
		// evtl. wait time if reset of device is necessary and then decide to go to states or ERROR state
		IF (CIf.Job.bolAlmReset = TRUE) THEN
			CIf.Job.eMe_ActivAlmClass := E_AlmClass.NONE; // reset feedback channel for parent
			CIf.Job.bolAlmReset := FALSE;
		END_IF
		
		// State Change Condition
		IF (CIf.Job.bolAlmReset = FALSE) THEN
			IF (me.StateMachine.intStateHistory<=BASE_PLC.cSTA_PON) THEN
				me.StateMachine.intStateNext := BASE_PLC.cSTA_PONBusy;
			END_IF;

			CASE me.intCmd OF
				BASE_PLC.cCMD_OFF:
					me.StateMachine.intStateNext := BASE_PLC.cSTA_OFFBusy;
				BASE_PLC.cCMD_RUN:
					me.StateMachine.intStateNext := BASE_PLC.cSTA_RUNBusy;
			ELSE
				CASE me.StateMachine.intStateHistory OF
					BASE_PLC.cSTA_RUN:
						me.StateMachine.intStateNext := BASE_PLC.cSTA_RUNBusy;
					BASE_PLC.cSTA_OFF:
						me.StateMachine.intStateNext := BASE_PLC.cSTA_OFFBusy;
					BASE_PLC.cSTA_STOP:
						me.StateMachine.intStateNext := BASE_PLC.cSTA_STOPBusy;
				END_CASE
			END_CASE
		END_IF
	END_IF




//--------------------------------------------------------------------------------------
// Exit action
	IF (me.StateMachine.intState<>me.StateMachine.intStateNext) THEN
		;
	END_IF
END_METHOD

{attribute 'object_name' := 'sta_OFF'}
METHOD PROTECTED sta_OFF : BOOL
// state implemetation
//--------------------------------------------------------------------------------------
// Entry action
	IF (me.StateMachine.intState<>me.StateMachine.intStateLastCycle) THEN
		me.StateMachine.intStateLastCycle := me.StateMachine.intState;
	END_IF


//--------------------------------------------------------------------------------------
// Cyclic action
	IF (me.StateMachine.intState=me.StateMachine.intStateLastCycle) THEN
		IF me.intCmd = BASE_PLC.cCMD_RUN THEN
			me.StateMachine.intStateNext := BASE_PLC.cSTA_RUNBusy;
		END_IF
	END_IF


//--------------------------------------------------------------------------------------
// Exit action
	IF (me.StateMachine.intState<>me.StateMachine.intStateNext) THEN
		;
	END_IF
END_METHOD

{attribute 'object_name' := 'sta_OFFBusy'}
METHOD PROTECTED sta_OFFBusy : BOOL
// state implemetation
//--------------------------------------------------------------------------------------
// Entry action
	IF (me.StateMachine.intState<>me.StateMachine.intStateLastCycle) THEN
		me.StateMachine.intStateLastCycle := me.StateMachine.intState;
		p_fbMotorIn^.CtrlCIf^.Job.intACmd := BASE_PLC.cCMD_OFF;
		p_fbMotorOut^.CtrlCIf^.Job.intACmd := BASE_PLC.cCMD_OFF;
		SIf.Out.bolVacuumValveIn.intern := FALSE;		
		SIf.Out.bolVacuumValveOut.intern := FALSE;		
	END_IF


//--------------------------------------------------------------------------------------
// Cyclic action
	IF (me.StateMachine.intState=me.StateMachine.intStateLastCycle) THEN
		IF p_fbMotorIn^.CtrlCIf^.Job.intState = BASE_PLC.cSTA_OFF 
		  AND p_fbMotorOut^.CtrlCIf^.Job.intState = BASE_PLC.cSTA_OFF THEN
			me.StateMachine.intStateNext := BASE_PLC.cSTA_OFF;
		END_IF
	END_IF


//--------------------------------------------------------------------------------------
// Exit action
	IF (me.StateMachine.intState<>me.StateMachine.intStateNext) THEN
		;
	END_IF
END_METHOD

{attribute 'object_name' := 'sta_PON'}
METHOD PROTECTED sta_PON : BOOL
// state implemetation
//--------------------------------------------------------------------------------------
// Entry action
	IF (me.StateMachine.intState<>me.StateMachine.intStateLastCycle) THEN
		me.StateMachine.intStateLastCycle := me.StateMachine.intState;
		
	END_IF


//--------------------------------------------------------------------------------------
// Cyclic action
	IF (me.StateMachine.intState=me.StateMachine.intStateLastCycle) THEN
		;
	END_IF




//--------------------------------------------------------------------------------------
// Exit action
	IF (me.StateMachine.intState<>me.StateMachine.intStateNext) THEN
		;
	END_IF
END_METHOD

{attribute 'object_name' := 'sta_RUN'}
METHOD PROTECTED sta_RUN : BOOL
VAR
	iDifference: INT;
END_VAR
// state implemetation
//--------------------------------------------------------------------------------------
// Entry action
	IF (me.StateMachine.intState<>me.StateMachine.intStateLastCycle) THEN
		me.StateMachine.intStateLastCycle := me.StateMachine.intState;
		
		IF SIf.In.bolPaperAvailable.intern THEN
			me.SubStateMachine.intStateNext := PCE_CmdState.cSUB_PAPEREXIT;
		ELSE
			me.SubStateMachine.intStateNext := PCE_CmdState.cSUB_PAPERENTRY;
		END_IF
	END_IF


//--------------------------------------------------------------------------------------
// Cyclic action
	IF (me.StateMachine.intState = me.StateMachine.intStateLastCycle) THEN
		CASE me.SubStateMachine.intState OF
			PCE_CmdState.cSUB_PAPERENTRY:
				PaperInputValveActive();
				
				IF SIf.In.bolPaperAvailable.intern THEN
					me.SubStateMachine.intStateNext := PCE_CmdState.cSUB_PAPERENTRYDelay;
				END_IF

				IF me.intCmd = BASE_PLC.cCMD_STOP THEN
					me.StateMachine.intStateNext := BASE_PLC.cSTA_STOPBusy;
				END_IF
			PCE_CmdState.cSUB_PAPERENTRYDelay:
				IF me.SubStateMachine.udiTimeInState_ms > SIf.Par.uinPaperEntryDelayTime_ms THEN
					me.SubStateMachine.intStateNext := PCE_CmdState.cSUB_PAPEREXIT;
				END_IF
			PCE_CmdState.cSUB_PAPEREXIT:
				PaperExitValveActive();

				IF NOT SIf.In.bolPaperAvailable.intern THEN
					me.SubStateMachine.intStateNext := PCE_CmdState.cSUB_PAPERENTRY;
				END_IF
				
				IF me.SubStateMachine.udiTimeInState_ms > SIf.Par.uinPaperExitTime_ms THEN
					pfbAlarmCtrl^.setAlarm(CIf.Info.intCtrlId,INT_TO_UINT(E_ALM_PCE.PaperSensorError),0,ADR(SIf.Alm),E_AlmState.RST,CIf.Job.eMe_ActivAlmClass);
					me.StateMachine.intStateNext := Base_PLC.cSTA_ERROR;	
				END_IF
		END_CASE
	END_IF


//--------------------------------------------------------------------------------------
// Exit action
	IF (me.StateMachine.intState<>me.StateMachine.intStateNext) THEN
		;
	END_IF
END_METHOD

{attribute 'object_name' := 'sta_RUNBusy'}
METHOD PROTECTED sta_RUNBusy : BOOL
// state implemetation
//--------------------------------------------------------------------------------------
// Entry action
	IF (me.StateMachine.intState<>me.StateMachine.intStateLastCycle) THEN
		me.StateMachine.intStateLastCycle := me.StateMachine.intState;
		p_fbMotorIn^.CtrlCIf^.Job.intACmd :=BASE_PLC.cCMD_RUN;
		p_fbMotorOut^.CtrlCIf^.Job.intACmd :=BASE_PLC.cCMD_RUN;
		
		IF SIf.In.bolPaperAvailable.intern THEN
			PaperExitValveActive();
		ELSE
			PaperInputValveActive();
		END_IF
	END_IF


//--------------------------------------------------------------------------------------
// Cyclic action
	IF (me.StateMachine.intState=me.StateMachine.intStateLastCycle) THEN
		IF (p_fbMotorIn^.CtrlCIf^.Job.intState = BASE_PLC.cSTA_RUN) 
		  AND (p_fbMotorOut^.CtrlCIf^.Job.intState = BASE_PLC.cSTA_RUN) THEN
			me.StateMachine.intStateNext := BASE_PLC.cSTA_RUN;
		END_IF

		IF me.intCmd = BASE_PLC.cCMD_STOP THEN
			me.StateMachine.intStateNext := BASE_PLC.cSTA_STOPBusy;
		END_IF
	END_IF


//--------------------------------------------------------------------------------------
// Exit action
	IF (me.StateMachine.intState<>me.StateMachine.intStateNext) THEN
		;
	END_IF
END_METHOD

{attribute 'object_name' := 'sta_STOP'}
METHOD PROTECTED sta_STOP : BOOL
// state implemetation
//--------------------------------------------------------------------------------------
// Entry action
	IF (me.StateMachine.intState<>me.StateMachine.intStateLastCycle) THEN
		me.StateMachine.intStateLastCycle := me.StateMachine.intState;
	END_IF


//--------------------------------------------------------------------------------------
// Cyclic action
	IF (me.StateMachine.intState=me.StateMachine.intStateLastCycle) THEN
		IF me.intCmd = BASE_PLC.cCMD_RUN THEN
			me.StateMachine.intStateNext := BASE_PLC.cSTA_RUNBusy;
		END_IF
	END_IF


//--------------------------------------------------------------------------------------
// Exit action
	IF (me.StateMachine.intState<>me.StateMachine.intStateNext) THEN
		;
	END_IF
END_METHOD

{attribute 'object_name' := 'sta_STOPBusy'}
METHOD PROTECTED sta_STOPBusy : BOOL
// state implemetation
//--------------------------------------------------------------------------------------
// Entry action
	IF (me.StateMachine.intState<>me.StateMachine.intStateLastCycle) THEN
		me.StateMachine.intStateLastCycle := me.StateMachine.intState;
		p_fbMotorIn^.CtrlCIf^.Job.intACmd := BASE_PLC.cCMD_STOP;
		p_fbMotorOut^.CtrlCIf^.Job.intACmd := BASE_PLC.cCMD_STOP;
	END_IF


//--------------------------------------------------------------------------------------
// Cyclic action
	IF (me.StateMachine.intState=me.StateMachine.intStateLastCycle) THEN
		IF p_fbMotorIn^.CtrlCIf^.Job.intState = BASE_PLC.cSTA_STOP 
		  AND p_fbMotorOut^.CtrlCIf^.Job.intState = BASE_PLC.cSTA_STOP  THEN
			me.StateMachine.intStateNext := BASE_PLC.cSTA_STOP;
		END_IF
	END_IF


//--------------------------------------------------------------------------------------
// Exit action
	IF (me.StateMachine.intState<>me.StateMachine.intStateNext) THEN
		;
	END_IF
END_METHOD

{attribute 'object_name' := 'StateMachine'}
METHOD PROTECTED StateMachine : BOOL
SUPER^.StateMachine();

// main statemachine of base controller
CASE me.StateMachine.intState OF
    BASE_PLC.cSTA_RUN: 
        THIS^.sta_RUN();
    BASE_PLC.cSTA_RUNBusy: 
        THIS^.sta_RUNBusy();
    BASE_PLC.cSTA_STOP: 
        THIS^.sta_STOP();
    BASE_PLC.cSTA_STOPBusy: 
        THIS^.sta_STOPBusy();
END_CASE;
END_METHOD

END_FUNCTION_BLOCK

// POUs/Controller/Lvl2/PST [Paper Stacker]/helper/cycle_Pst
FUNCTION cycle_Pst : BOOL
VAR_INPUT
	pPst: POINTER TO T_PST;
END_VAR

pPst^.ctrl.fbPst_Ptb_Umc.In_bolEmoOk 				:= pPst^.io.In_bolPtb_Umc_EmoOk;
pPst^.ctrl.fbPst_Ptb_Umc.In_uinStatus 				:= pPst^.io.In_uinPtb_Umc_Status;
pPst^.ctrl.fbPst_Ptb_Umc.In_intMotorActualSpeed 	:= pPst^.io.In_uinPtb_Umc_ActualSpeed;
pPst^.ctrl.fbPst_Ptb_Umc.In_uinMotorSetSpeed 		:= pPst^.io.In_uinPtb_Umc_SetSpeed;
pPst^.ctrl.fbPst_Ptb_Umc.In_uinECATState 			:= pPst^.io.In_uinPtb_Umc_ECatState;
pPst^.ctrl.fbPst_Ptb_Umc.In_strNetId 				:= pPst^.io.In_strPtb_Umc_ECatNetId;
pPst^.ctrl.fbPst_Ptb_Umc.In_uintPort 				:= pPst^.io.In_uinPtb_Umc_ECatPort;
pPst^.ctrl.fbPst_Ptb_Umc();
pPst^.io.Out_uinPtb_Umc_SetSpeed 					:= pPst^.ctrl.fbPst_Ptb_Umc.Out_uinSpeedSetpoint;
pPst^.io.Out_uinPtb_Umc_Control 					:= pPst^.ctrl.fbPst_Ptb_Umc.Out_uinControl;

pPst^.ctrl.fbPst_Ptb_Vpc.In_bolPumpOk 				:= pPst^.io.In_bolPtb_Vpc_PumpOk;
pPst^.ctrl.fbPst_Ptb_Vpc.In_bolVacuumOk 			:= pPst^.io.In_bolPtb_Vpc_VacuumSensor;
pPst^.ctrl.fbPst_Ptb_Vpc();
pPst^.io.Out_bolPtb_Vpc_PumpOn 						:= pPst^.ctrl.fbPst_Ptb_Vpc.Out_bolVaccumPumpOn;

pPst^.ctrl.fbPst_Ptb.In_bolBeltEntrySensor		 	:= pPst^.io.In_bolPtb_InputSensor;
pPst^.ctrl.fbPst_Ptb.In_bolBeltExitSensor 			:= pPst^.io.In_bolPtb_OutputSensor;
pPst^.ctrl.fbPst_Ptb();

pPst^.ctrl.fbPst.In_bolSensorPaperAtOperatorPos		:= pPst^.io.In_bolSensorPaperAtOperatorPos;
pPst^.ctrl.fbPst.In_bolSensorStopperPosition		:= pPst^.io.In_bolSensorStopperPosition;
pPst^.ctrl.fbPst.In_bolSensorInfeed					:= pPst^.io.In_bolSensorInfeed;
pPst^.ctrl.fbPst.In_bolSensorOutfeed				:= pPst^.io.In_bolSensorOutfeed;
pPst^.ctrl.fbPst();

END_FUNCTION

// POUs/Controller/Lvl2/PST [Paper Stacker]/helper/init_Pst
FUNCTION init_Pst : BOOL
VAR_INPUT
	pPst			: POINTER TO T_PST;
	/// instance array of all controller instances
	pCtrlInst		: POINTER TO fb_CtrlBase;
	/// common interface array of all controllers (main use for PLC)
	pCtrlCIf		: POINTER TO T_Ctrl_CIf;
END_VAR

pPst^.ctrl.fbPst_Ptb_Vpc.iniAllCtrlArrays(pCtrlInst,pCtrlCIf,pPst^.id.Pst_Ptb_Vpc);
pPst^.ctrl.fbPst_Ptb_Umc.iniAllCtrlArrays(pCtrlInst,pCtrlCIf,pPst^.id.Pst_Ptb_Umc);
pPst^.ctrl.fbPst_Ptb.iniAllCtrlArrays(pCtrlInst,pCtrlCIf,pPst^.id.Pst_Ptb);
pPst^.ctrl.fbPst_Ptb.Drive := ADR(pPst^.ctrl.fbPst_Ptb_Umc); // g_a_pCtrlInst[pPst^.id.Pst_Ptb_Umc];
pPst^.ctrl.fbPst_Ptb.VacuumPump := ADR(pPst^.ctrl.fbPst_Ptb_Vpc); // g_a_pCtrlInst[pPst^.id.Pst_Ptb_Vpc];

pPst^.ctrl.fbPst.iniAllCtrlArrays(pCtrlInst,pCtrlCIf,pPst^.id.Pst);
pPst^.ctrl.fbPst.Belt := ADR(pPst^.ctrl.fbPst_Ptb);; // g_a_pCtrlInst[pPst^.id.Pst_Ptb];

END_FUNCTION

// POUs/Controller/Lvl2/PST [Paper Stacker]/FB_PST
FUNCTION_BLOCK FB_PST EXTENDS FB_CtrlBase
VAR_INPUT
	In_uinBarcodeEvent: UINT;
	In_ulnBarcode: ULINT;
	In_bolSensorPaperAtOperatorPos: BOOL;
	In_bolSensorStopperPosition: BOOL;
	In_bolSensorInfeed: BOOL;
	In_bolSensorOutfeed: BOOL;
END_VAR
VAR
	/// Specific interface struct for public access
	SIf: T_Ctrl_SIf_PST;
	/// Paper stacker belt
	p_fbBelt: POINTER TO FB_PTB;
	pBeltCIf: POINTER TO T_Ctrl_CIf;
	pBeltSif: POINTER TO T_Ctrl_SIf_PTB;
	/// Variables for edge detection
	bolSensorInfeedOld: BOOL;
	bolSensorOutfeedOld: BOOL;
	uinStackHightOld: UINT;
	/// Tmp. Barcode reader data
	stBarcodeData: T_BCC_Data;
	/// Retry counter
	uinRetryCounter: UINT;
	/// Simulation
	udiSimTimerPaperInfeedStroke: UDINT;
	/// Data Channel to saber for paper stack info
	p_fbPaperStackFifo: POINTER TO FB_DataChannelSenderFifo;
END_VAR

(*__________________________________________________________________________________________________
¦	
¦	Vistaprint Schweiz GmbH
¦	CH - 8401 Winterthur
¦
¦	www.vistaprint.ch - info@vistaprint.ch
¦___________________________________________________________________________________________________

Function desription:
...

History:
Version		Date			Author		Comment
---------------------------------------------------------------------------------------------------
0.00.1		23.06.2014		AVME/DSC	Start history
___________________________________________________________________________________________________*)


SUPER^();

{attribute 'object_name' := 'Always'}
METHOD PROTECTED Always : BOOL
SUPER^.Always();

// ----------------------------------------------------------------------------------
// cyclic actions outside of statemachine
IF (me.StateMachine.intState<>cSTA_SINGLE_ANSWER) THEN
	
	// Simulation
	// --------------------------------------------
	IF (CIf.SwCfg.bolSimulation) THEN
		// Simulate a new paper at infeed
		IF (me.StateMachine.intState = Base_PLC.cSTA_RUN) AND (me.SubStateMachine.intState = PST_CmdState.cSUB_WAITNEWPAPERDETECTED) AND (me.StateMachine.intState <> PST_CmdState.cSTA_EJECTbusy) THEN
			IF (udiSimTimerPaperInfeedStroke >= SIf.Par.udiSimTimePaperInfeedStroke_ms) THEN
				SIf.In.bolSensorInfeed.intern:= TRUE;
			END_IF
		ELSE
			udiSimTimerPaperInfeedStroke:= 0;
			SIf.In.bolSensorInfeed.intern:= FALSE;		
		END_IF			
		// Timer handling
		udiSimTimerPaperInfeedStroke:= udiSimTimerPaperInfeedStroke + me.FUBInfo.udiSample_ms;
	ELSE
		udiSimTimerPaperInfeedStroke:= 0;
	END_IF
	
	
	// Single paper infeed counting
	// --------------------------------------------
	// Inc. stack hight with every pos. edge of infeed sensor 
	IF (SIf.In.bolSensorInfeed.intern) AND NOT (bolSensorInfeedOld) THEN
		SIf.Cur.uinStackHight:= SIf.Cur.uinStackHight + 1;
	END_IF
	bolSensorInfeedOld:= SIf.In.bolSensorInfeed.intern;
			
	// Monitoring of special error conditions
	// --------------------------------------------
	
	// If a new paper is detected at the feeding during the ejection -> Alarm!
	IF (me.StateMachine.intState = PST_CmdState.cSTA_EJECTbusy) THEN
		// New paper detected/counted 
		IF (SIf.Cur.uinStackHight <> uinStackHightOld) AND NOT (SIf.Cur.bolStackIncomplete) THEN
			SIf.Cur.bolStackIncomplete:= TRUE;
			pfbAlarmCtrl^.setAlarm(CIf.Info.intCtrlId,E_ALM_PST.NewPaperDetectedDuringEjecting,0,ADR(SIf.Alm),E_AlmState.RST,CIf.Job.eMe_ActivAlmClass);
		END_IF	
	END_IF	
	
	// If a new paper is detected at the feeding while barcode reading process -> Alarm!				
	IF (me.StateMachine.intState = Base_PLC.cSTA_RUN) AND (me.SubStateMachine.intState <> PST_CmdState.cSUB_WAITNEWPAPERDETECTED) THEN
		// New paper detected/counted 
		IF (SIf.Cur.uinStackHight <> uinStackHightOld) AND NOT (SIf.Cur.bolStackIncomplete) THEN
			SIf.Cur.bolStackIncomplete:= TRUE;
			pfbAlarmCtrl^.setAlarm(CIf.Info.intCtrlId,E_ALM_PST.NewPaperDetectedWhileBarcodeReading,0,ADR(SIf.Alm),E_AlmState.RST,CIf.Job.eMe_ActivAlmClass);
		END_IF
	END_IF
			
END_IF

// ----------------------------------------------------------------------------------
// Always change actions in Base Library
// ----------------------------------------------------------------------------------
// overrule error always from base -> no EOFF State!! in EOFF go to OFF
IF (me.StateMachine.intStateNext = cSTA_EOFFBusy) THEN
	IF (me.StateMachine.intState=cSTA_OFF) THEN
		me.StateMachine.intStateNext := cSTA_OFF;
	ELSE // stay in OFF
		me.StateMachine.intStateNext := cSTA_OFFBusy;
	END_IF
END_IF

// Conditions Always
IF (((me.Alarm.eActivAlmClass=E_AlmClass.EOFF) OR (me.Alarm.eActivAlmClass=E_AlmClass.OFF) OR (me.intCmd=cCMD_OFF))
		 AND (me.StateMachine.intState<>cSTA_ERROR) AND (me.StateMachine.intState<>cSTA_ERRORQuit) AND
		(me.StateMachine.intState<>cSTA_OFF) AND (me.StateMachine.intState<>cSTA_OFFBusy) AND (me.StateMachine.intState<>cSTA_SINGLE_ANSWER)) THEN
	// alarm evt EOFF, OFF or cmd off
	me.StateMachine.intStateNext := cSTA_OFFBusy;
END_IF
END_METHOD

PROPERTY Belt : POINTER TO FB_PTB
GET
Belt := p_fbBelt;
END_GET
SET
p_fbBelt := Belt;
END_SET
END_PROPERTY

{attribute 'object_name' := 'CtrlInit'}
METHOD CtrlInit : BOOL
SUPER^.CtrlInit();

pBeltCIf := p_fbBelt^.CtrlCIf;
pBeltSIf := p_fbBelt^.getCtrlSIf();

AddChild(p_fbBelt^);

// Initialize stack buffer
IF (p_fbPaperStackFifo <> TC3_MEMMAN.NULL) THEN
	p_fbPaperStackFifo^.FreeDataPointer := TRUE;
	p_fbPaperStackFifo^.Enable := TRUE;
END_IF
END_METHOD

PROPERTY PUBLIC CtrlSIf : POINTER TO T_Ctrl_SIf_PST
GET
CtrlSIf := ADR(SIf);
END_GET
END_PROPERTY

{attribute 'object_name' := 'FB_init'}
METHOD FB_init : BOOL
VAR_INPUT
	/// if TRUE, the retain variables are initialized (warm start / cold start)
	bInitRetains: BOOL;
	/// if TRUE, the instance afterwards gets moved into the copy code (online change)
	bInCopyCode: BOOL;
END_VAR
VAR
	iIdx: UINT;
	iLength: UINT;
END_VAR
//------------------------------------------------------------------------------------------------------------------------
// to manually change in new FUB implementation!!!
// define valid commands for this controller
iLength := SIZEOF(CIf.Job.aCmdList)/SIZEOF(CIf.Job.aCmdList[0]);
iIdx := 0;

WHILE (iIdx < iLength) AND (CIf.Job.aCmdList[iIdx].intCmd <> cCMD_INITIALIZED) DO
	iIdx := iIdx + 1; 
END_WHILE

IF (iIdx < iLength) THEN
// Add configuration of own comands	
	CIf.Job.aCmdList[iIdx].intCmd := BASE_PLC.cCMD_RUN;
	CIf.Job.aCmdList[iIdx].strName := 'RUN'; 
	CIf.Job.aCmdList[iIdx].bolAvailable := TRUE;
	iIdx := iIdx + 1;
	CIf.Job.aCmdList[iIdx].intCmd := PST_CmdState.cCMD_EJECT;
	CIf.Job.aCmdList[iIdx].strName := 'EJECT'; 
	CIf.Job.aCmdList[iIdx].bolAvailable := TRUE;
ELSE
	// Error if the aCmdList Array is to small
END_IF

// set name of class/typ
CIf.Info.strType := 'FB_PST';
CIf.Info.strFullName := 'Paper Stacker';

// set alarm class

SIf.Alm[E_ALM_PST.StackIncomplete].eAlmClass := Base_PLC.E_AlmClass.TSTOP;
SIf.Alm[E_ALM_PST.StackIncomplete].strText := 'Stack incomplete. Stacker was sent to OFF before finishing the job!';
SIf.Alm[E_ALM_PST.NeedsEjectCommand].eAlmClass := Base_PLC.E_AlmClass.WARNING;
SIf.Alm[E_ALM_PST.NeedsEjectCommand].strText := 'Last job was incomplete. Stacker waits for an eject command!';
SIf.Alm[E_ALM_PST.StackOkButLastCodeNotRight].eAlmClass := Base_PLC.E_AlmClass.OFF;
SIf.Alm[E_ALM_PST.StackOkButLastCodeNotRight].strText := 'Stack hight is reached but last barcode ID is not right!';
SIf.Alm[E_ALM_PST.StackNotOkButLastCodeRight].eAlmClass := Base_PLC.E_AlmClass.OFF;
SIf.Alm[E_ALM_PST.StackNotOkButLastCodeRight].strText := 'Stack hight is not reached but last barcode ID is right!';
SIf.Alm[E_ALM_PST.ReadingBarcodeFailedAfterXRetries].eAlmClass := Base_PLC.E_AlmClass.OFF;
SIf.Alm[E_ALM_PST.ReadingBarcodeFailedAfterXRetries].strText := 'Reading barcode failed after X retries!';
SIf.Alm[E_ALM_PST.NewPaperDetectedDuringEjecting].eAlmClass := Base_PLC.E_AlmClass.OFF;
SIf.Alm[E_ALM_PST.NewPaperDetectedDuringEjecting].strText := 'New paper detected during ejecting is in process!';
SIf.Alm[E_ALM_PST.NewPaperDetectedWhileBarcodeReading].eAlmClass := Base_PLC.E_AlmClass.OFF;
SIf.Alm[E_ALM_PST.NewPaperDetectedWhileBarcodeReading].strText := 'New paper detected while barcode reading is in process!';

//*******************************************************************************
// initial values
//*******************************************************************************

// software configuration
CIf.SwCfg.bolExist := TRUE;
CIf.SwCfg.bolEnable := TRUE;
CIf.SwCfg.bolSimulation := FALSE;

// Configuration
SIf.Cfg.bolEnableDataChannel:= FALSE;
SIf.Cfg.uinNumOfRetryRead:= 3;
SIf.Cfg.usiEjectingDirection:= E_BELT_DIRECTION.FORWARD; // Right
SIf.Cfg.usiReverseDirection:= E_BELT_DIRECTION.BACKWARD; // Left
SIf.Cfg.bolEnablePstEjectControl := FALSE;

// parameter
SIf.Par.uinStackHight:= 0;
SIf.Par.uliLastBarCodeInStack:= 0;

SIf.Par.uinBeltReverseSpeed_mmsec:= 250; 
SIf.Par.uinBeltEjectSpeed_mmsec:= 300;
SIf.Par.udiPaperAtOpPosDebounceTime_ms:= 1000;
SIf.Par.udiStopperPosDebounceTime_ms:= 1000;
SIf.Par.udiSensorOutfeedDebounceTime_ms:= 1000;
SIf.Par.udiStackEjectDelayTime_ms:= 1000;
SIf.Par.udiBeltReverseDelayTime_ms:= 1000;
SIf.Par.udiStackEjectingTime_ms:= 4000;
SIf.Par.udiBarcodeReaderTriggerDelayTime_ms:= 1500;
SIf.Par.udiSimTimePaperInfeedStroke_ms:= 5000;
END_METHOD

{attribute 'object_name' := 'getCmdState'}
METHOD PROTECTED getCmdState : STRING
VAR_INPUT
	intCmdState: INT;
	bolState: BOOL;
END_VAR
getCmdState := SUPER^.getCmdState(intCmdState:=intCmdState,bolState:=bolState); // get global/base defined cmds/states

IF (getCmdState='') THEN // global not defined get local
	// get string cmd/state string information in runtime
	IF (bolState=FALSE) THEN
		CASE intCmdState OF
			PST_CmdState.cCMD_EJECT:
				getCmdState := 'EJECT';
		END_CASE;
	ELSE
		// States's
		CASE intCmdState OF
			PST_CmdState.cSTA_EJECTbusy: 
				getCmdState := 'EJECTbusy';
			
			// sub states	
			PST_CmdState.cSUB_WAITNEWPAPERDETECTED: 
				getCmdState := 'WAITNEWPAPERDETECTED';	
			PST_CmdState.cSUB_DELAYREADBARCODEBusy: 
				getCmdState := 'DELAYREADBARCODEBusy';	
			PST_CmdState.cSUB_RETRYREADBARCODE: 
				getCmdState := 'RETRYREADBARCODE';	
			PST_CmdState.cSUB_READBARCODEbusy: 
				getCmdState := 'READBARCODEbusy';	
			PST_CmdState.cSUB_CHECKEJECTCONDITIONS: 
				getCmdState := 'CHECKEJECTCONDITIONS';	
			
			PST_CmdState.cSUB_DELAYSTACKEJECTBusy: 
				getCmdState := 'DELAYSTACKEJECTBusy';	
			PST_CmdState.cSUB_MOVEBELTEJECTDIRECTIONBusy: 
				getCmdState := 'MOVEBELTEJECTDIRECTIONBusy';	
			PST_CmdState.cSUB_STOPBELTBusy: 
				getCmdState := 'STOPBELTBusy';	
			PST_CmdState.cSUB_WAITBEFOREMOVINGREVERSE: 
				getCmdState := 'WAITBEFOREMOVINGREVERSE';	
			PST_CmdState.cSUB_MOVEBELTREVERSEBusy: 
				getCmdState := 'MOVEBELTREVERSEBusy';		
										
			PST_CmdState.cSUB_DONE: 
				getCmdState := 'DONE';	
		END_CASE;
	END_IF
END_IF
END_METHOD

{attribute 'object_name' := 'getCtrlSIf'}
METHOD getCtrlSIf : POINTER TO T_Ctrl_SIf_PST
getCtrlSIf := ADR(SIf);
END_METHOD

{attribute 'object_name' := 'IoInBridge'}
METHOD PROTECTED IoInBridge : BOOL
// digitale and analoge inputs read from hardware or forcing
SIf.In.bolSensorPaperAtOperatorPos.map := THIS^.In_bolSensorPaperAtOperatorPos;
SIf.In.bolSensorStopperPosition.map := THIS^.In_bolSensorStopperPosition;
SIf.In.bolSensorInfeed.map := THIS^.In_bolSensorInfeed;
SIf.In.bolSensorOutfeed.map := THIS^.In_bolSensorOutfeed;

IF (CIf.SwCfg.bolSimulation = FALSE) THEN
	getInBolDebounced(CIf.Job.bolIoForce,me.FUBInfo.udiSample_ms, sif.Par.udiPaperAtOpPosDebounceTime_ms,  ADR(SIf.In.bolSensorPaperAtOperatorPos));
	getInBolDebounced(CIf.Job.bolIoForce,me.FUBInfo.udiSample_ms, sif.Par.udiStopperPosDebounceTime_ms,  ADR(SIf.In.bolSensorStopperPosition));	
	getInBolDebounced(CIf.Job.bolIoForce,me.FUBInfo.udiSample_ms, sif.Par.udiSensorOutfeedDebounceTime_ms, ADR(SIf.In.bolSensorOutfeed));
	getInBol(CIf.Job.bolIoForce,ADR(SIf.In.bolSensorInfeed));
ELSE
	;//simulation of global IO
END_IF
END_METHOD

PROPERTY PaperStackSendFifo : POINTER TO FB_DataChannelSenderFifo
SET
p_fbPaperStackFifo := PaperStackSendFifo;
END_SET
END_PROPERTY

{attribute 'object_name' := 'sta_EJECTBusy'}
METHOD PROTECTED sta_EJECTBusy : BOOL
// state implemetation
//--------------------------------------------------------------------------------------
// Entry action
	IF (me.StateMachine.intState<>me.StateMachine.intStateLastCycle) THEN
		me.StateMachine.intStateLastCycle := me.StateMachine.intState;
		
		CIf.Job.intACmd:= Base_PLC.cCMD_DONE;
		CIf.Job.intMCmd:= Base_PLC.cCMD_DONE;

		SIf.Cur.bolStackIncomplete:= TRUE;
		
		// Initialize sub state machine
		me.SubStateMachine.intState:= PST_CmdState.cSUB_DELAYSTACKEJECTBusy; 
		me.SubStateMachine.intStateNext:= PST_CmdState.cSUB_DELAYSTACKEJECTBusy;	
	END_IF

//--------------------------------------------------------------------------------------
// Cyclic action
	IF (me.StateMachine.intState=me.StateMachine.intStateLastCycle) THEN
			
		// ---------------------------------------------------------
		// Sub state machine for handling ejecting the paper stack
		// ---------------------------------------------------------
		CASE me.SubStateMachine.intState OF
		
			// Wait before moving in eject direction
			PST_CmdState.cSUB_DELAYSTACKEJECTBusy:
				// Entry action
				IF (me.SubStateMachine.intState<>me.SubStateMachine.intStateLastCycle) THEN
					me.SubStateMachine.intStateLastCycle := me.SubStateMachine.intState;		
				END_IF
			
				// Wait X time before starting the belt
				IF (me.SubStateMachine.udiTimeInState_ms >= SIf.Par.udiStackEjectDelayTime_ms) THEN
					// Start the belt
					pBeltSif^.Par.intDirection := SIf.Cfg.usiEjectingDirection;
					pBeltSif^.Par.rBeltParam.uinBeltSpeed:= SIf.Par.uinBeltEjectSpeed_mmsec;					
					p_fbBelt^.CIf.Job.intACmd:= cCMD_RUN;
					me.SubStateMachine.intStateNext := PST_CmdState.cSUB_MOVEBELTEJECTDIRECTIONBusy;	
				END_IF
				
			// Belt is moving in eject direction
			PST_CmdState.cSUB_MOVEBELTEJECTDIRECTIONBusy:
				// Entry action
				IF (me.SubStateMachine.intState<>me.SubStateMachine.intStateLastCycle) THEN
					me.SubStateMachine.intStateLastCycle := me.SubStateMachine.intState;		
				END_IF
				
				// Simulation
				// --------------------------------------------
				IF (CIf.SwCfg.bolSimulation) THEN
					// stopper is in down position
					SIf.In.bolSensorStopperPosition.intern:= FALSE;
				END_IF
		
				// Wait until stack ejecting time expired and stopper is in down position
				IF (me.SubStateMachine.udiTimeInState_ms >= SIf.Par.udiStackEjectingTime_ms) AND (NOT SIf.In.bolSensorStopperPosition.intern) THEN
					// Wait until paper stack has left outfeed sensor position
					IF NOT (SIf.In.bolSensorOutfeed.intern) THEN
						// Stop belt
						p_fbBelt^.Cif.Job.intACmd:= cCMD_STOP;
						me.SubStateMachine.intStateNext := PST_CmdState.cSUB_STOPBELTBusy;
					END_IF	
				END_IF
		
			// Wait before moving in reverse direction
			PST_CmdState.cSUB_WAITBEFOREMOVINGREVERSE:
				// Entry action
				IF (me.SubStateMachine.intState<>me.SubStateMachine.intStateLastCycle) THEN
					me.SubStateMachine.intStateLastCycle := me.SubStateMachine.intState;		
				END_IF
				
				// Wait X time before starting the belt in reverse direction
				IF (me.SubStateMachine.udiTimeInState_ms >= SIf.Par.udiBeltReverseDelayTime_ms) THEN
					// Start the belt
					pBeltSif^.Par.intDirection := SIf.Cfg.usiReverseDirection;
					pBeltSif^.Par.rBeltParam.uinBeltSpeed:= SIf.Par.uinBeltReverseSpeed_mmsec;
					p_fbBelt^.Cif.Job.intACmd:= cCMD_RUN;
					me.SubStateMachine.intStateNext := PST_CmdState.cSUB_MOVEBELTREVERSEBusy;	
				END_IF
				
			// Belt is moving in reverse direction
			PST_CmdState.cSUB_MOVEBELTREVERSEBusy:
				// Entry action
				IF (me.SubStateMachine.intState<>me.SubStateMachine.intStateLastCycle) THEN
					me.SubStateMachine.intStateLastCycle := me.SubStateMachine.intState;		
				END_IF
				
				// Simulation
				// --------------------------------------------
				IF (CIf.SwCfg.bolSimulation) THEN
					// stopper is in down position
					SIf.In.bolSensorStopperPosition.intern:= TRUE;
				END_IF
			
				// Wait until stopper is in up position
				IF (SIf.In.bolSensorStopperPosition.intern) THEN
					// Stop belt
					p_fbBelt^.Cif.Job.intACmd:= cCMD_STOP;
					me.SubStateMachine.intStateNext := PST_CmdState.cSUB_STOPBELTBusy;	
				END_IF
					
			// Stop belt busy
			PST_CmdState.cSUB_STOPBELTBusy:
				
				// Wait until belt stopped
				IF (p_fbBelt^.Cif.Job.intState = Base_PLC.cSTA_STOP) THEN
					// Decision dependent last cycle state
					IF (me.SubStateMachine.intStateLastCycle = PST_CmdState.cSUB_MOVEBELTEJECTDIRECTIONBusy) THEN
						// Go on with wait before moving reverse
						me.SubStateMachine.intStateNext := PST_CmdState.cSUB_WAITBEFOREMOVINGREVERSE;
					ELSE	
						// Done
						me.SubStateMachine.intStateNext := PST_CmdState.cSUB_DONE;
					END_IF
				END_IF
				
			// All done
			PST_CmdState.cSUB_DONE:
				// Entry action
				IF (me.SubStateMachine.intState<>me.SubStateMachine.intStateLastCycle) THEN
					me.SubStateMachine.intStateLastCycle := me.SubStateMachine.intState;		
				END_IF

				SIf.Cur.bolStackIncomplete:= FALSE;
				SIf.Par.uinStackHight:= 0;
				// Update counter stacks ejected total
				SIf.Cur.udiNumOfStacksEjectedTotal:= SIf.Cur.udiNumOfStacksEjectedTotal + 1;
				// Back to RUN!
				me.StateMachine.intStateNext := Base_PLC.cSTA_RUNBusy;	
				
		END_CASE	
	
	END_IF

//--------------------------------------------------------------------------------------
// Exit action
	IF (me.StateMachine.intState<>me.StateMachine.intStateNext) THEN
		;
	END_IF
END_METHOD

{attribute 'object_name' := 'sta_OFF'}
METHOD PROTECTED sta_OFF : BOOL
// state implemetation
//--------------------------------------------------------------------------------------
// Entry action
	IF (me.StateMachine.intState<>me.StateMachine.intStateLastCycle) THEN
		me.StateMachine.intStateLastCycle := me.StateMachine.intState;
		CIf.Job.intACmd:= Base_PLC.cCMD_DONE;
		CIf.Job.intMCmd:= Base_PLC.cCMD_DONE;
	END_IF

//--------------------------------------------------------------------------------------
// Cyclic action
	IF (me.StateMachine.intState=me.StateMachine.intStateLastCycle) THEN
		
		CASE me.intCmd OF
			
			// Command RUN	
			BASE_PLC.cCMD_RUN:
				me.StateMachine.intStateNext := BASE_PLC.cSTA_RUNBusy;
				
			// Command EJECT	
			PST_CmdState.cCMD_EJECT:
				me.StateMachine.intStateNext := PST_CmdState.cSTA_EJECTbusy;
				
		END_CASE

	END_IF

//--------------------------------------------------------------------------------------
// Exit action
	IF (me.StateMachine.intState<>me.StateMachine.intStateNext) THEN
		;
	END_IF
END_METHOD

{attribute 'object_name' := 'sta_OFFBusy'}
METHOD PROTECTED sta_OFFBusy : BOOL
// state implemetation
//--------------------------------------------------------------------------------------
// Entry action
	IF (me.StateMachine.intState<>me.StateMachine.intStateLastCycle) THEN
		me.StateMachine.intStateLastCycle := me.StateMachine.intState;
	
		IF (p_fbPaperStackFifo <> TC3_MEMMAN.NULL) THEN
			// Enable data channel
			p_fbPaperStackFifo^.Enable := SIf.Cfg.bolEnableDataChannel;
			// Clear buffer
			p_fbPaperStackFifo^.ClearFifo();
		END_IF
		
		// Childs off
		p_fbBelt^.CtrlCIf^.Job.intACmd := BASE_PLC.cCMD_OFF;
	
		// In case of an OFF command or alarm, check if the stack is incomplete. 
		// Only check if min. stack hight of 1 paper is set by saber
		IF ((SIf.Cur.uinStackHight <> SIf.Par.uinStackHight) AND (SIf.Par.uinStackHight >= 1) AND NOT (SIf.Cur.bolStackIncomplete)) OR NOT SIf.In.bolSensorStopperPosition.intern THEN
			// Stack incomplete! Saber has to send an eject command before next RUN.
			SIf.Cur.bolStackIncomplete:= TRUE;
			pfbAlarmCtrl^.setAlarm(CIf.Info.intCtrlId,E_ALM_PST.StackIncomplete,0,ADR(SIf.Alm),E_AlmState.RST,CIf.Job.eMe_ActivAlmClass);
		ELSE
			// ... do nothing, normal scenario!		
		END_IF
	
	END_IF

//--------------------------------------------------------------------------------------
// Cyclic action
	IF (me.StateMachine.intState=me.StateMachine.intStateLastCycle) THEN
		
		IF (p_fbBelt^.CtrlCIf^.Job.intState = BASE_PLC.cSTA_OFF)  THEN 
			me.StateMachine.intStateNext := BASE_PLC.cSTA_OFF;
		END_IF	
	END_IF

//--------------------------------------------------------------------------------------
// Exit action
	IF (me.StateMachine.intState<>me.StateMachine.intStateNext) THEN
		;
	END_IF
END_METHOD

{attribute 'object_name' := 'sta_RUN'}
METHOD PROTECTED sta_RUN : BOOL
VAR
	pItemPaperInfo: POINTER TO T_ItemPaperInfo;
END_VAR
// state implemetation
//--------------------------------------------------------------------------------------
// Entry action
IF (me.StateMachine.intState<>me.StateMachine.intStateLastCycle) THEN
	me.StateMachine.intStateLastCycle := me.StateMachine.intState;
	// Initialize sub state machine
	me.SubStateMachine.intState:= PST_CmdState.cSUB_WAITNEWPAPERDETECTED; 
	me.SubStateMachine.intStateNext:= PST_CmdState.cSUB_WAITNEWPAPERDETECTED;	
END_IF

//--------------------------------------------------------------------------------------
// Cyclic action
IF (me.StateMachine.intState = me.StateMachine.intStateLastCycle) THEN
	
	// -------------------------------------------------------------------------------
	// Sub state machine for reading barcode and make decision for ejecting the stack
	// -------------------------------------------------------------------------------
	CASE me.SubStateMachine.intState OF
	
		// Wait until new paper was detected at stacker infeed position
		PST_CmdState.cSUB_WAITNEWPAPERDETECTED:
		
			// New paper detected/counted 
			IF (SIf.Cur.uinStackHight <> uinStackHightOld) THEN
				uinStackHightOld:= SIf.Cur.uinStackHight;
				
				IF SIf.Cfg.bolEnablePstEjectControl THEN
					me.SubStateMachine.intStateNext := PST_CmdState.cSUB_CHECKEJECTCONDITIONS;
				END_IF
			END_IF
		
			CASE me.intCmd OF
				// Command EJECT	
				PST_CmdState.cCMD_EJECT:
					me.StateMachine.intStateNext := PST_CmdState.cSTA_EJECTbusy;
			END_CASE

		// Check the eject conditions after successful read
		PST_CmdState.cSUB_CHECKEJECTCONDITIONS:
		
			// Check if the stack hight is reached and last barcode ID is right
			IF (SIf.Cur.uinStackHight = SIf.Par.uinStackHight) AND (stBarcodeData.uliBarCode = SIf.Par.uliLastBarCodeInStack) THEN
				// Stack complete!
				// New job can be sent by saber!
//				SIf.Par.uinStackHight:= 0;
				SIf.Par.uliLastBarCodeInStack:= 0;
				// Done -> EJECT stack
				me.SubStateMachine.intStateNext := PST_CmdState.cSUB_DONE;
			ELSE
				// Stack not complete -> wait for next paper
				me.SubStateMachine.intStateNext := PST_CmdState.cSUB_WAITNEWPAPERDETECTED;
			END_IF
		
			// Error conditions
			// -------------------------
			
			// Stack hight is reached but last barcode ID is not right!
			IF (SIf.Cur.uinStackHight = SIf.Par.uinStackHight) AND (stBarcodeData.uliBarCode <> SIf.Par.uliLastBarCodeInStack) THEN				
				SIf.Cur.bolStackIncomplete:= TRUE;
				pfbAlarmCtrl^.setAlarm(CIf.Info.intCtrlId,E_ALM_PST.StackOkButLastCodeNotRight,0,ADR(SIf.Alm),E_AlmState.RST,CIf.Job.eMe_ActivAlmClass);
			END_IF
		
			// Stack hight is not reached but last barcode ID is right!
			IF (SIf.Cur.uinStackHight <> SIf.Par.uinStackHight) AND (stBarcodeData.uliBarCode = SIf.Par.uliLastBarCodeInStack) THEN
				SIf.Cur.bolStackIncomplete:= TRUE;
				pfbAlarmCtrl^.setAlarm(CIf.Info.intCtrlId,E_ALM_PST.StackNotOkButLastCodeRight,0,ADR(SIf.Alm),E_AlmState.RST,CIf.Job.eMe_ActivAlmClass);
			END_IF

		// All done
		PST_CmdState.cSUB_DONE:
			me.StateMachine.intStateNext := PST_CmdState.cSTA_EJECTbusy;	
			
	END_CASE	

END_IF


//--------------------------------------------------------------------------------------
// Exit action
IF (me.StateMachine.intState<>me.StateMachine.intStateNext) THEN
	;
END_IF
END_METHOD

{attribute 'object_name' := 'sta_RUNBusy'}
METHOD PROTECTED sta_RUNBusy : BOOL
// state implemetation
//--------------------------------------------------------------------------------------
// Entry action
	IF (me.StateMachine.intState<>me.StateMachine.intStateLastCycle) THEN
		me.StateMachine.intStateLastCycle := me.StateMachine.intState;
		CIf.Job.intACmd:= Base_PLC.cCMD_DONE;
		CIf.Job.intMCmd:= Base_PLC.cCMD_DONE;
		// Clear stack hight
		SIf.Cur.uinStackHight:= 0;
		uinStackHightOld:= 0;		
	END_IF


//--------------------------------------------------------------------------------------
// Cyclic action
	IF (me.StateMachine.intState=me.StateMachine.intStateLastCycle) THEN
		
		IF SIf.Cur.bolStackIncomplete THEN
			pfbAlarmCtrl^.setAlarm(CIf.Info.intCtrlId,E_ALM_PST.NeedsEjectCommand,0,ADR(SIf.Alm),E_AlmState.RST,CIf.Job.eMe_ActivAlmClass);
			me.StateMachine.intStateNext := PST_CmdState.cSTA_EJECTbusy;
		ELSE
			me.StateMachine.intStateNext := BASE_PLC.cSTA_RUN;
		END_IF
	END_IF

//--------------------------------------------------------------------------------------
// Exit action
	IF (me.StateMachine.intState<>me.StateMachine.intStateNext) THEN
		;
	END_IF
END_METHOD

{attribute 'object_name' := 'StateMachine'}
METHOD PROTECTED StateMachine : BOOL
SUPER^.StateMachine();

// main statemachine of base controller
CASE me.StateMachine.intState OF
    BASE_PLC.cSTA_RUN: 
        THIS^.sta_RUN();
    BASE_PLC.cSTA_RUNBusy: 
        THIS^.sta_RUNBusy();
	PST_CmdState.cSTA_EJECTbusy:
        THIS^.sta_EJECTBusy();
END_CASE;
END_METHOD

END_FUNCTION_BLOCK

// POUs/Controller/Lvl2/PTS [Paper Turning Station]/helper/cycle_Pts
FUNCTION cycle_Pts : BOOL
VAR_INPUT
	pPts: POINTER TO T_PTS;
END_VAR

pPts^.ctrl.fbPts_Ptb_Umc.In_bolEmoOk 				:= pPts^.io.In_bolPtb_Umc_EmoOk;
pPts^.ctrl.fbPts_Ptb_Umc.In_uinStatus 				:= pPts^.io.In_uinPtb_Umc_Status;
pPts^.ctrl.fbPts_Ptb_Umc.In_intMotorActualSpeed		:= pPts^.io.In_uinPtb_Umc_ActualSpeed;
pPts^.ctrl.fbPts_Ptb_Umc.In_uinMotorSetSpeed		:= pPts^.io.In_uinPtb_Umc_SetSpeed;
pPts^.ctrl.fbPts_Ptb_Umc.In_uinECATState 			:= pPts^.io.In_uinPtb_Umc_ECatState;
pPts^.ctrl.fbPts_Ptb_Umc.In_strNetId 				:= pPts^.io.In_strPtb_Umc_ECatNetId;
pPts^.ctrl.fbPts_Ptb_Umc.In_uintPort 				:= pPts^.io.In_uinPtb_Umc_ECatPort;
pPts^.ctrl.fbPts_Ptb_Umc();
pPts^.io.Out_uinPtb_Umc_SetSpeed 					:= pPts^.ctrl.fbPts_Ptb_Umc.Out_uinSpeedSetpoint;
pPts^.io.Out_uinPtb_Umc_Control 					:= pPts^.ctrl.fbPts_Ptb_Umc.Out_uinControl;

pPts^.ctrl.fbPts_Ptb_Vpc.In_bolPumpOk 				:= pPts^.io.In_bolPtb_Vpc_PumpOk;
pPts^.ctrl.fbPts_Ptb_Vpc.In_bolVacuumOk 			:= pPts^.io.In_bolPtb_Vpc_VacuumSensor;
pPts^.ctrl.fbPts_Ptb_Vpc();
pPts^.io.Out_bolPtb_Vpc_PumpOn 						:= pPts^.ctrl.fbPts_Ptb_Vpc.Out_bolVaccumPumpOn;

IF (pPts^.ctrl.fbPts.CtrlSIf^.Cfg.bolRaxEnable = FALSE) THEN
	pPts^.ctrl.fbPts_Mdc_Umc.In_bolEmoOk 				:= pPts^.io.In_bolMdc_Umc_EmoOk;
	pPts^.ctrl.fbPts_Mdc_Umc.In_uinStatus 				:= pPts^.io.In_uinMdc_Umc_Status;
	pPts^.ctrl.fbPts_Mdc_Umc.In_intMotorActualSpeed		:= pPts^.io.In_uinMdc_Umc_ActualSpeed;
	pPts^.ctrl.fbPts_Mdc_Umc.In_uinMotorSetSpeed 		:= pPts^.io.In_uinMdc_Umc_SetSpeed;
	pPts^.ctrl.fbPts_Mdc_Umc.In_uinECATState 			:= pPts^.io.In_uinMdc_Umc_ECatState;
	pPts^.ctrl.fbPts_Mdc_Umc.In_strNetId 				:= pPts^.io.In_strMdc_Umc_ECatNetId;
	pPts^.ctrl.fbPts_Mdc_Umc.In_uintPort 				:= pPts^.io.In_uinMdc_Umc_ECatPort;
	pPts^.ctrl.fbPts_Mdc_Umc();
	pPts^.io.Out_uinMdc_Umc_SetSpeed 					:= pPts^.ctrl.fbPts_Mdc_Umc.Out_uinSpeedSetpoint;
	pPts^.io.Out_uinMdc_Umc_Control 					:= pPts^.ctrl.fbPts_Mdc_Umc.Out_uinControl;
	
	pPts^.ctrl.fbPts_Mdc.In_bolCrossPositionSensor 		:= pPts^.io.In_bolMdc_CrossPositionSensor;
	pPts^.ctrl.fbPts_Mdc.In_bolTablePositionSensor 		:= pPts^.io.In_bolMdc_TablePositionSensor;
	pPts^.ctrl.fbPts_Mdc();
ELSE
	pPts^.ctrl.fbPts_RAX_POD.In_bolHomeSwitch			:= pPts^.io.In_bolRax_PositionSensor;
	pPts^.ctrl.fbPts_RAX_POD();

	pPts^.ctrl.fbPts_RAX();
END_IF

pPts^.ctrl.fbPts_Ptb();

pPts^.ctrl.fbPts.In_bol_PaperAvailable 				:= pPts^.io.In_bolPaperSensor;
pPts^.ctrl.fbPts();

END_FUNCTION

// POUs/Controller/Lvl2/PTS [Paper Turning Station]/helper/init_Pts
FUNCTION init_Pts : BOOL
VAR_INPUT
	pPts			: POINTER TO T_PTS;
	/// instance array of all controller instances
	pCtrlInst		: POINTER TO fb_CtrlBase;
	/// common interface array of all controllers (main use for PLC)
	pCtrlCIf		: POINTER TO T_Ctrl_CIf;
END_VAR

pPts^.ctrl.fbPts_Ptb_Vpc.iniAllCtrlArrays(pCtrlInst,pCtrlCIf,pPts^.id.Pts_Ptb_Vpc);
pPts^.ctrl.fbPts_Ptb_Umc.iniAllCtrlArrays(pCtrlInst,pCtrlCIf,pPts^.id.Pts_Ptb_Umc);
pPts^.ctrl.fbPts_Ptb.iniAllCtrlArrays(pCtrlInst,pCtrlCIf,pPts^.id.Pts_Ptb);
pPts^.ctrl.fbPts_Ptb.Drive := ADR(pPts^.ctrl.fbPts_Ptb_Umc);
pPts^.ctrl.fbPts_Ptb.VacuumPump := ADR(pPts^.ctrl.fbPts_Ptb_Vpc);

pPts^.ctrl.fbPts_Mdc_Umc.iniAllCtrlArrays(pCtrlInst,pCtrlCIf,pPts^.id.Pts_Mdc_Umc);
pPts^.ctrl.fbPts_Mdc.iniAllCtrlArrays(pCtrlInst,pCtrlCIf,pPts^.id.Pts_Mdc);
pPts^.ctrl.fbPts_Mdc.Drive := ADR(pPts^.ctrl.fbPts_Mdc_Umc);

pPts^.ctrl.fbPts_RAX.iniAllCtrlArrays(pCtrlInst,pCtrlCIf,pPts^.id.Pts_RAX);
pPts^.ctrl.fbPts_RAX.In_pAD_SIf:= pPts^.ctrl.fbPts_RAX_POD.AD_SIf;	

pPts^.ctrl.fbPts.iniAllCtrlArrays(pCtrlInst,pCtrlCIf,pPts^.id.Pts);
pPts^.ctrl.fbPts.Belt := ADR(pPts^.ctrl.fbPts_Ptb);
pPts^.ctrl.fbPts.Malteser := ADR(pPts^.ctrl.fbPts_Mdc);
pPts^.ctrl.fbPts.Servo := ADR(pPts^.ctrl.fbPts_RAX);

END_FUNCTION

// POUs/Controller/Lvl2/PTS [Paper Turning Station]/FB_PTS
FUNCTION_BLOCK FB_PTS EXTENDS FB_CtrlBase
VAR_INPUT
	In_bol_PaperAvailable: BOOL;
	In_bol_PaperAtBeltExit: BOOL;
END_VAR
VAR
	/// Specific interface struct for public access
	SIf: T_Ctrl_SIf_PTS;
	///pointer to function block
	p_fbBelt: POINTER TO FB_PTB;
	pBeltCIf: POINTER TO BASE_PLC.T_Ctrl_CIf;
	p_fbMalteser: POINTER TO FB_MDC;
	pMalteserCIf: POINTER TO BASE_PLC.T_Ctrl_CIf;
	/// Rotary Axis instead of Malteser
	p_fbRAX: POINTER TO FB_RAX;
	/// Rotary Axis instead of Malteser
	pRaxCIf: POINTER TO BASE_PLC.T_Ctrl_CIf;
	bolPrePositionBusy: BOOL;
	intActualPosition: INT;
	intTargetPosition: INT;
	/// Position to go to if comand turn is given. 0 = initialization position, 1, 2, 3
	uinPositionToGo: UINT;
	/// <0 = Turn left; =0 automatic; >0 turn right
	intTurnDirection: INT;
END_VAR

(*__________________________________________________________________________________________________
¦	
¦	Vistaprint Schweiz GmbH
¦	CH - 8401 Winterthur
¦
¦	www.vistaprint.ch - info@vistaprint.ch
¦___________________________________________________________________________________________________

Function desription:
Destacker/Buffer implementation. 


History:
Version		Date			Author		Comment
---------------------------------------------------------------------------------------------------
0.00.1		09.07.2013		PC			Start history
0.00.2		24.09.2014		AVME/MRU	Servo instead of MCD added
0.00.3		19.11.2014		AVME/MRU	Changes after Commissioning
0.00.4		12.12.2014		AVME/MRU	Connect Input of HomeSensor
0.00.5		16.12.2014		AVME/MRU	Add long term test
___________________________________________________________________________________________________*)


IF (me.bolActivate) THEN // cyclic call enabled
	IF (CIf.Info.bolInitDone=FALSE) THEN // first cycle -> init
		CtrlInit();
		CIf.Info.bolInitDone := TRUE;
	ELSE
		CycleStartDuty();
	
		Always();
		
		StateMachine();

		CycleEndDuty();
	END_IF
END_IF;

{attribute 'object_name' := 'Always'}
METHOD PROTECTED Always : BOOL
SUPER^.Always();

// ----------------------------------------------------------------------------------
// cyclic actions outside of statemachine
IF (me.StateMachine.intState<>cSTA_SINGLE_ANSWER) THEN
	
	; // always error supervision
	
END_IF

// ----------------------------------------------------------------------------------
// Conditions Always
IF (((me.Alarm.eActivAlmClass=E_AlmClass.EOFF) OR (me.Alarm.eActivAlmClass=E_AlmClass.OFF) OR (me.intCmd=cCMD_OFF) OR (me.intCmd=BASE_PLC.cCMD_EOFF))
		 AND (me.StateMachine.intState<>cSTA_ERROR) AND (me.StateMachine.intState<>cSTA_ERRORQuit) AND
		(me.StateMachine.intState<>cSTA_OFF) AND (me.StateMachine.intState<>cSTA_OFFBusy)) THEN
	// alarm evt EOFF, OFF or cmd off
	me.StateMachine.intStateNext := cSTA_OFFBusy;
END_IF

IF SIf.Cfg.bolRaxEnable THEN
	IF pRaxCIf = NULL THEN
		SIf.Cfg.bolRaxEnable := FALSE;
		pfbAlarmCtrl^.setAlarm(CIf.Info.intCtrlId,INT_TO_UINT(E_ALM_PTS.TurnTableConfigMissmatch),0,ADR(SIf.Alm),E_AlmState.RST,CIf.Job.eMe_ActivAlmClass);
	END_IF
ELSE
	IF pMalteserCIf = NULL THEN
		SIf.Cfg.bolRaxEnable := TRUE;
		pfbAlarmCtrl^.setAlarm(CIf.Info.intCtrlId,INT_TO_UINT(E_ALM_PTS.TurnTableConfigMissmatch),0,ADR(SIf.Alm),E_AlmState.RST,CIf.Job.eMe_ActivAlmClass);
	END_IF
END_IF

SIf.Cur.udiPTS_Counter := udiPTS_Counter_Persistent;		// Update SIf.Cur Variable
END_METHOD

PROPERTY Belt : POINTER TO FB_PTB
GET
Belt := p_fbBelt;
END_GET
SET
p_fbBelt := Belt;
END_SET
END_PROPERTY

{attribute 'object_name' := 'CalculateOutputDelay'}
METHOD PRIVATE CalculateOutputDelay : UDINT
VAR_INPUT
	uinBeltSpeed: UINT;
	udiInputDelay: UDINT;
END_VAR
VAR
	relBeltSpeed: LREAL;
	relInputDelay: LREAL;
END_VAR
relBeltSpeed := UINT_TO_REAL(uinBeltSpeed);
relInputDelay := UDINT_TO_LREAL(udiInputDelay);
CalculateOutputDelay := LREAL_TO_UDINT((1000.0*(750.0 - ((relBeltSpeed/1000)*(750.0+relInputDelay))))/relBeltSpeed);
END_METHOD

{attribute 'object_name' := 'ChangeDistributionModeParameter'}
METHOD ChangeDistributionModeParameter : BOOL
VAR_INPUT
	eMode: E_PTS_MODE;
	uinBeltSpeed: UINT;
	uinRotationSpeed: UINT;
END_VAR
SIf.Par.eMode := eMode;
p_fbBelt^.CtrlSIf^.Par.rBeltParam.uinBeltSpeed := uinBeltSpeed;		
IF (SIf.Cfg.bolRaxEnable) THEN
	p_fbRAX^.CtrlSIf^.Par.dinSpeed_0_1deg_s := uinRotationSpeed;
ELSE
	p_fbMalteser^.Drive^.CtrlSIf^.Par.uinSpeed_rpm := uinRotationSpeed;
END_IF
END_METHOD

{attribute 'object_name' := 'CtrlInit'}
METHOD CtrlInit : BOOL
SUPER^.CtrlInit();

IF (SIf.Cfg.bolRaxEnable) THEN
	THIS^.AddChild(p_fbRAX^);

	pRaxCIf := p_fbRAX^.CtrlCIf;
ELSE
	THIS^.AddChild(p_fbMalteser^);

	pMalteserCIf := p_fbMalteser^.CtrlCIf;
END_IF

THIS^.AddChild(p_fbBelt^);

pBeltCIf := p_fbBelt^.CtrlCIf;

(*
// set parent id
pMalteserCIf^.Info.intParentCtrlId := CIf.Info.intCtrlId;			
pBeltCIf^.Info.intParentCtrlId := CIf.Info.intCtrlId;			

//necessary???
THIS^.CIf.Info.p_aCIf[0] := pMalteserCIf;
THIS^.CIf.Info.p_aCIf[1] := pBeltCIf;
*)
END_METHOD

PROPERTY PUBLIC CtrlSIf : POINTER TO T_Ctrl_SIf_PTS
GET
CtrlSIf := ADR(SIf);
END_GET
END_PROPERTY

{attribute 'object_name' := 'FB_init'}
METHOD FB_init : BOOL
VAR_INPUT
	/// if TRUE, the retain variables are initialized (warm start / cold start)
	bInitRetains: BOOL;
	/// if TRUE, the instance afterwards gets moved into the copy code (online change)
	bInCopyCode: BOOL;
END_VAR
VAR
	iIdx: UINT;
	iLength: UINT;
END_VAR
//------------------------------------------------------------------------------------------------------------------------
// to manually change in new FUB implementation!!!
// define valid commands for this controller
iLength := SIZEOF(CIf.Job.aCmdList)/SIZEOF(CIf.Job.aCmdList[0]);
iIdx := 0;

WHILE (iIdx < iLength) AND (CIf.Job.aCmdList[iIdx].intCmd <> cCMD_INITIALIZED) DO
	iIdx := iIdx + 1; 
END_WHILE

IF (iIdx < iLength) THEN
// Add configuration of own comands	
	CIf.Job.aCmdList[iIdx].intCmd := BASE_PLC.cCMD_RUN;
	CIf.Job.aCmdList[iIdx].strName := 'RUN'; 
	CIf.Job.aCmdList[iIdx].bolAvailable := TRUE;
	iIdx := iIdx + 1;
	CIf.Job.aCmdList[iIdx].intCmd := BASE_PLC.cCMD_STOP;
	CIf.Job.aCmdList[iIdx].strName := 'STOP'; 
	CIf.Job.aCmdList[iIdx].bolAvailable := TRUE;
	iIdx := iIdx + 1;
	CIf.Job.aCmdList[iIdx].intCmd := PTS_CmdState.cCMD_STANDBY;
	CIf.Job.aCmdList[iIdx].strName := 'STANDBY'; 
	CIf.Job.aCmdList[iIdx].bolAvailable := TRUE;
	iIdx := iIdx + 1;
	CIf.Job.aCmdList[iIdx].intCmd := PTS_CmdState.cCMD_TURN;
	CIf.Job.aCmdList[iIdx].strName := 'TURN'; 
	CIf.Job.aCmdList[iIdx].bolAvailable := TRUE;
ELSE
	// Error if the aCmdList Array is to small
END_IF

// set name of class/typ
CIf.Info.strType := 'FB_PTS'; 
CIf.Info.strFullName := 'Paper Turning Station';

// set alarm class
SIf.Alm[E_ALM_PTS.PaperTransport].eAlmClass := E_AlmClass.TSTOP;
SIf.Alm[E_ALM_PTS.PaperTransport].strText := 'Possible Paper Jam';
SIf.Alm[E_ALM_PTS.ModeParameter].eAlmClass := E_AlmClass.TSTOP;
SIf.Alm[E_ALM_PTS.ModeParameter].strText := 'Wrong Mode Parameter';
SIf.Alm[E_ALM_PTS.TurnTableConfigMissmatch].eAlmClass := E_AlmClass.WARNING;
SIf.Alm[E_ALM_PTS.TurnTableConfigMissmatch].strText := 'Turn Table Type Configuration Missmatch';

//*******************************************************************************
// initial values
//*******************************************************************************

// software configuration
CIf.SwCfg.bolExist := TRUE;
CIf.SwCfg.bolEnable := TRUE;
CIf.SwCfg.bolSimulation := FALSE;

// configuration
SIf.Cfg.bolPositionMalteserEnable := TRUE;

// parameter
SIf.Cfg.bolBarcodeReaderAvailable := FALSE;
SIf.Cfg.aDefaultAutoPos := 0;
SIf.Cfg.aFixPosDef[E_PTS_MODE.FixA].uinInput := 0;
SIf.Cfg.aFixPosDef[E_PTS_MODE.FixA].uinOutput := 1;
SIf.Cfg.aFixPosDef[E_PTS_MODE.FixB].uinInput := 3;
SIf.Cfg.aFixPosDef[E_PTS_MODE.FixB].uinOutput := 2;
SIf.Cfg.aFixPosDef[E_PTS_MODE.FixC].uinInput := 0;
SIf.Cfg.aFixPosDef[E_PTS_MODE.FixC].uinOutput := 0;
SIf.Cfg.aAutoPosDef[0].uinInput := 0;
SIf.Cfg.aAutoPosDef[0].uinOutput := 0;
SIf.Cfg.aAutoPosDef[1].uinInput := 0;
SIf.Cfg.aAutoPosDef[1].uinOutput := 1;
SIf.Cfg.aDistributionPositionDefinition[0] := E_PTS_MODE.FixC; 
SIf.Cfg.aDistributionPositionDefinition[1] := E_PTS_MODE.FixA; 
SIf.Cfg.bolRaxEnable := True;		// Use Servo Axis instead of Malteser 
SIf.Par.eMode := E_PTS_MODE.FixC;
SIf.Par.udiPaperBarcodeToInputSensorTime := 2000;
SIf.Par.udiPaperInTurnDelayTime := 000;
SIf.Par.udiPaperOutTurnDelayTime := 300;
SIf.Par.udiSimPaperBarcodeToInputSensorTime := SIf.Par.udiPaperBarcodeToInputSensorTime / 2;
SIf.Par.bolLongTimeTestEnable := False;
END_METHOD

{attribute 'object_name' := 'getCmdState'}
METHOD PROTECTED getCmdState : STRING
VAR_INPUT
	intCmdState: INT;
	bolState: BOOL;
END_VAR
getCmdState := SUPER^.getCmdState(intCmdState:=intCmdState,bolState:=bolState); // get global/base defined cmds/states

IF (getCmdState='') THEN // global not defined get local
	// get string cmd/state string information in runtime
	IF (bolState=FALSE) THEN
		CASE intCmdState OF
			PTS_CmdState.cCMD_STANDBY: 
				getCmdState := 'cCMD_STANDBY';
			PTS_CmdState.cCMD_TURN: 
				getCmdState := 'cCMD_TURN';
		END_CASE;
	ELSE
		// States's
		CASE intCmdState OF
			PTS_CmdState.cSTA_EmptyDelayBusy: 
				getCmdState := 'cSTA_EmptyDelayBusy';
			PTS_CmdState.cSTA_GetItemBusy: 
				getCmdState := 'cSTA_GetItemBusy';
			PTS_CmdState.cSTA_InitializeBusy: 
				getCmdState := 'cSTA_InitializeBusy';
			PTS_CmdState.cSTA_PaperDelayBusy: 
				getCmdState := 'cSTA_PaperDelayBusy';
			PTS_CmdState.cSTA_STANDBY: 
				getCmdState := 'cSTA_STANDBY';
			PTS_CmdState.cSTA_STANDBYBusy: 
				getCmdState := 'cSTA_STANDBYBusy';
			PTS_CmdState.cSTA_TurnEmptyBusy: 
				getCmdState := 'cSTA_TurnEmptyBusy';
			PTS_CmdState.cSTA_TurnPaperBusy: 
				getCmdState := 'cSTA_TurnPaperBusy';
			PTS_CmdState.cSTA_WaitPaper: 
				getCmdState := 'cSTA_WaitPaper';
			PTS_CmdState.cSTA_WaitPaperGone: 
				getCmdState := 'cSTA_WaitPaperGone';
		END_CASE;
	END_IF
END_IF
END_METHOD

{attribute 'object_name' := 'getCtrlSIf'}
METHOD getCtrlSIf : POINTER TO T_Ctrl_SIf_PTS
getCtrlSIf := ADR(SIf);
END_METHOD

{attribute 'object_name' := 'GetItemBusy'}
METHOD PROTECTED GetItemBusy : BOOL
END_METHOD

{attribute 'object_name' := 'IoInBridge'}
METHOD PROTECTED IoInBridge : BOOL
// digitale and analoge inputs read from hardware or forcing
SIf.In.bolPaperAvailable.map			:= NOT THIS^.In_bol_PaperAvailable;
SIf.In.bolPaperAtBeltExit.map			:= THIS^.In_bol_PaperAtBeltExit;

IF (CIf.SwCfg.bolSimulation = FALSE) THEN
	BASE_PLC.getInBol(CIf.Job.bolIoForce,ADR(SIf.In.bolPaperAvailable));
	BASE_PLC.getInBol(CIf.Job.bolIoForce,ADR(SIf.In.bolPaperAtBeltExit));
ELSE
	SIf.In.bolPaperAvailable.map		:= FALSE;
	BASE_PLC.getInBol(CIf.Job.bolIoForce,ADR(SIf.In.bolPaperAvailable));
END_IF
END_METHOD

{attribute 'object_name' := 'IoOutBridge'}
METHOD PROTECTED IoOutBridge : BOOL
VAR
	bolSwitchValvesOff: BOOL;
END_VAR
// digitale and analoge inputs read from hardware or forcing
IF (CIf.SwCfg.bolSimulation = FALSE) THEN
	;
END_IF

// Write Outputs to Turning Child (Malteser or ServoDrive)
IF (SIf.Cfg.bolRaxEnable) THEN
	// ToDo: p_fbRAX^.CtrlSIf^.Par. intTurnDirection := intTurnDirection;
	p_fbRAX^.CtrlSIf^.Par.dinPos_0_1Deg := uinPositionToGo*90*10;	
ELSE
	p_fbMalteser^.CtrlSIf^.Par.intTurnDirection := intTurnDirection;	// <0 = Turn left; =0 automatic; >0 turn right
	p_fbMalteser^.CtrlSIf^.Par.uinPositionToGo := uinPositionToGo;
END_IF
END_METHOD

PROPERTY Malteser : POINTER TO FB_MDC
GET
Malteser := p_fbMalteser;
END_GET
SET
p_fbMalteser := Malteser;
END_SET
END_PROPERTY

PROPERTY Servo : POINTER TO FB_MDC
GET
Servo := p_fbRAX;
END_GET
SET
p_fbRAX := Servo;
END_SET
END_PROPERTY

{attribute 'object_name' := 'sta_ERROR'}
METHOD PROTECTED sta_ERROR : BOOL
// state implemetation
//--------------------------------------------------------------------------------------
// Entry action
	IF (me.StateMachine.intState<>me.StateMachine.intStateLastCycle) THEN
		me.StateMachine.intStateHistory := me.StateMachine.intStateLastCycle; // -> possibillity to go back to state before error
		me.StateMachine.intStateLastCycle := me.StateMachine.intState;
		
		// stop child controllers
		pBeltCIf^.Job.intACmd := BASE_PLC.cCMD_OFF;
		IF (SIf.Cfg.bolRaxEnable) THEN
			pRaxCIf^.Job.intACmd := cCMD_OFF;
		ELSE
			pMalteserCIf^.Job.intACmd := BASE_PLC.cCMD_OFF;
		END_IF
	END_IF


//--------------------------------------------------------------------------------------
// Cyclic action
	IF (me.StateMachine.intState=me.StateMachine.intStateLastCycle) THEN
		
		;
		
		
		// State Change Condition
		IF (CIf.Job.bolAlmReset = TRUE) THEN
			me.StateMachine.intStateNext := cSTA_ERRORQuit;
		END_IF
	END_IF




//--------------------------------------------------------------------------------------
// Exit action
	IF (me.StateMachine.intState<>me.StateMachine.intStateNext) THEN
		;
	END_IF
END_METHOD

{attribute 'object_name' := 'sta_ERRORQuit'}
METHOD PROTECTED sta_ERRORQuit : BOOL
// state implemetation
//--------------------------------------------------------------------------------------
// Entry action
	IF (me.StateMachine.intState<>me.StateMachine.intStateLastCycle) THEN
		me.StateMachine.intStateLastCycle := me.StateMachine.intState;
		
	END_IF


//--------------------------------------------------------------------------------------
// Cyclic action
	IF (me.StateMachine.intState=me.StateMachine.intStateLastCycle) THEN
		
		;
		// evtl. wait time if reset of device is necessary and then decide to go to states or ERROR state
		IF (CIf.Job.bolAlmReset = TRUE) THEN
			CIf.Job.eMe_ActivAlmClass := E_AlmClass.NONE; // reset feedback channel for parent
			CIf.Job.bolAlmReset := FALSE;
		END_IF
		
		// State Change Condition
		IF (CIf.Job.bolAlmReset = FALSE) THEN
			IF (me.StateMachine.intStateHistory<=cSTA_PON) THEN
				me.StateMachine.intStateNext := cSTA_PONBusy;
			ELSE
				IF me.intCmd >= 0 THEN
					CASE me.intCmd OF
						cCMD_OFF:
							me.StateMachine.intStateNext := cSTA_OFFBusy;
						cCMD_RUN:
							me.StateMachine.intStateNext := cSTA_RUNBusy;
						cCMD_STOP:
							me.StateMachine.intStateNext := cSTA_STOPBusy;
					END_CASE
				ELSE
					CASE me.StateMachine.intStateHistory OF
						cSTA_PaperDelayBusy,cSTA_TurnPaperBusy,
						cSTA_WaitPaperGone,cSTA_EmptyDelayBusy,
						cSTA_TurnEmptyBusy,cSTA_WaitPaper,
						cSTA_RUNBusy, cSTA_RUN:
							me.StateMachine.intStateNext := cSTA_RUNBusy;
					ELSE
						me.StateMachine.intStateNext := cSTA_OFFBusy;
					END_CASE
				END_IF
			END_IF
		END_IF
	END_IF




//--------------------------------------------------------------------------------------
// Exit action
	IF (me.StateMachine.intState<>me.StateMachine.intStateNext) THEN
		;
	END_IF
END_METHOD

{attribute 'object_name' := 'sta_GetItemBusy'}
METHOD PROTECTED sta_GetItemBusy : BOOL
END_METHOD

{attribute 'object_name' := 'sta_InitializeBusy'}
METHOD PROTECTED sta_InitializeBusy : BOOL
// state implemetation
//--------------------------------------------------------------------------------------
// Entry action
	IF (me.StateMachine.intState<>me.StateMachine.intStateLastCycle) THEN
		me.StateMachine.intStateLastCycle := me.StateMachine.intState;
		IF (SIf.Cfg.bolRaxEnable) THEN
			pRaxCIf^.Job.intACmd := cCMD_INIT;
		ELSE
			pMalteserCIf^.Job.intACmd := MDC_CmdState.cCMD_INITIALIZE;
		END_IF
	END_IF


//--------------------------------------------------------------------------------------
// Cyclic action
	IF (me.StateMachine.intState=me.StateMachine.intStateLastCycle) THEN
		IF (SIf.Cfg.bolRaxEnable) THEN
			IF (pRaxCIf^.Job.intState = cSTA_INIT) THEN
				pRaxCIf^.Job.intACmd := cCMD_STOP;				
				me.StateMachine.intStateNext := PTS_CmdState.cSTA_STANDBYBusy;
			END_IF
		ELSE
			IF (pMalteserCIf^.Job.intState = MDC_CmdState.cSTA_InPosition) THEN
				me.StateMachine.intStateNext := PTS_CmdState.cSTA_STANDBYBusy;
			END_IF
		END_IF
	END_IF


//--------------------------------------------------------------------------------------
// Exit action
	IF (me.StateMachine.intState<>me.StateMachine.intStateNext) THEN
		;
	END_IF
END_METHOD

{attribute 'object_name' := 'sta_OFF'}
METHOD PROTECTED sta_OFF : BOOL
// state implemetation
//--------------------------------------------------------------------------------------
// Entry action
	IF (me.StateMachine.intState<>me.StateMachine.intStateLastCycle) THEN
		me.StateMachine.intStateLastCycle := me.StateMachine.intState;

	END_IF


//--------------------------------------------------------------------------------------
// Cyclic action
	IF (me.StateMachine.intState=me.StateMachine.intStateLastCycle) THEN
		CASE me.intCmd OF
			BASE_PLC.cCMD_RUN,
			PTS_CmdState.cCMD_STANDBY,
			Base_plc.cCMD_STOP: 
				me.StateMachine.intStateNext := PTS_CmdState.cSTA_InitializeBusy;
		END_CASE
	END_IF


//--------------------------------------------------------------------------------------
// Exit action
	IF (me.StateMachine.intState<>me.StateMachine.intStateNext) THEN
		;
	END_IF
END_METHOD

{attribute 'object_name' := 'sta_OFFBusy'}
METHOD PROTECTED sta_OFFBusy : BOOL
// state implemetation
//--------------------------------------------------------------------------------------
// Entry action
	IF (me.StateMachine.intState<>me.StateMachine.intStateLastCycle) THEN
		me.StateMachine.intStateLastCycle := me.StateMachine.intState;
		pBeltCIf^.Job.intACmd := BASE_PLC.cCMD_OFF;
		IF (SIf.Cfg.bolRaxEnable) THEN
			pRaxCIf^.Job.intACmd := cCMD_OFF;
		ELSE
			pMalteserCIf^.Job.intACmd := BASE_PLC.cCMD_OFF;
		END_IF
		SIf.Cur.iActualDistributionIndex := 0;
	END_IF


//--------------------------------------------------------------------------------------
// Cyclic action
	IF (me.StateMachine.intState=me.StateMachine.intStateLastCycle) THEN
		IF (SIf.Cfg.bolRaxEnable) THEN
			IF (pBeltCIf^.Job.intState = BASE_PLC.cSTA_OFF) AND (pRaxCIf^.Job.intState = BASE_PLC.cSTA_OFF) THEN
				me.StateMachine.intStateNext := BASE_PLC.cSTA_OFF;
			END_IF
		ELSE			
			IF (pBeltCIf^.Job.intState = BASE_PLC.cSTA_OFF) AND (pMalteserCIf^.Job.intState = BASE_PLC.cSTA_OFF) THEN
				me.StateMachine.intStateNext := BASE_PLC.cSTA_OFF;
			END_IF
		END_IF
	END_IF


//--------------------------------------------------------------------------------------
// Exit action
	IF (me.StateMachine.intState<>me.StateMachine.intStateNext) THEN
		;
	END_IF
END_METHOD

{attribute 'object_name' := 'sta_PaperDelayBusy'}
METHOD PROTECTED sta_PaperDelayBusy : BOOL
// state implemetation
//--------------------------------------------------------------------------------------
// Entry action
	IF (me.StateMachine.intState<>me.StateMachine.intStateLastCycle) THEN
		me.StateMachine.intStateLastCycle := me.StateMachine.intState;
//		Log Message ---------------------
		TC2_SYSTEM.ADSLOGSTR(ADSLOG_MSGTYPE_LOG,'%s','sta_PaperDelayBusy');
//		---------------------------------
	END_IF


//--------------------------------------------------------------------------------------
// Cyclic action
	IF (me.StateMachine.intState = me.StateMachine.intStateLastCycle) THEN
		IF (me.StateMachine.udiTimeInState_ms > SIf.Par.udiPaperInTurnDelayTime) THEN
			me.StateMachine.intStateNext := PTS_CmdState.cSTA_TurnPaperBusy;
		END_IF
	END_IF


//--------------------------------------------------------------------------------------
// Exit action
	IF (me.StateMachine.intState<>me.StateMachine.intStateNext) THEN
		;
	END_IF
END_METHOD

{attribute 'object_name' := 'sta_PON'}
METHOD PROTECTED sta_PON : BOOL
// state implemetation
//--------------------------------------------------------------------------------------
// Entry action
	IF (me.StateMachine.intState<>me.StateMachine.intStateLastCycle) THEN
		me.StateMachine.intStateLastCycle := me.StateMachine.intState;
		
	END_IF


//--------------------------------------------------------------------------------------
// Cyclic action
	IF (me.StateMachine.intState=me.StateMachine.intStateLastCycle) THEN
		;
	END_IF




//--------------------------------------------------------------------------------------
// Exit action
	IF (me.StateMachine.intState<>me.StateMachine.intStateNext) THEN
		;
	END_IF
END_METHOD

{attribute 'object_name' := 'sta_RUN'}
METHOD PROTECTED sta_RUN : BOOL
// state implemetation
//--------------------------------------------------------------------------------------
// Entry action
	IF (me.StateMachine.intState<>me.StateMachine.intStateLastCycle) THEN
		me.StateMachine.intStateLastCycle := me.StateMachine.intState;
		CIf.Job.intACmd := BASE_PLC.cCMD_DONE;
		CIf.Job.intMCmd := BASE_PLC.cCMD_DONE;
	END_IF


//--------------------------------------------------------------------------------------
// Cyclic action
	IF (me.StateMachine.intState = me.StateMachine.intStateLastCycle) THEN
		CASE SIf.Par.eMode OF
			E_PTS_MODE.Automatic:
				pfbAlarmCtrl^.setAlarm(CIf.Info.intCtrlId,INT_TO_UINT(E_ALM_PTS.ModeParameter),0,ADR(SIf.Alm),E_AlmState.RST,CIf.Job.eMe_ActivAlmClass);
	(*
				IF SIf.Cfg.bolBarcodeReaderAvailable (* AND BCR has a new barcode read *) THEN
					me.StateMachine.intStateNext := PTS_CmdState.cSTA_GetItemBusy;
				ELSE
					pfbAlarmCtrl^.setAlarm(CIf.Info.intCtrlId,INT_TO_UINT(E_ALM_PTS.ModeParameter),0,ADR(SIf.Alm),E_AlmState.RST,CIf.Job.eMe_ActivAlmClass);
				END_IF
	*)
			E_PTS_MODE.Distribute:
				IF ((NOT SIf.Cfg.bolEntrySensorAvailable) OR (SIf.In.bolPaperAtBeltExit.intern)) THEN
//					SIf.Cur.rInOutPosition := SIf.Cfg.aFixPosDef[SIf.Cfg.aDistributionPositionDefinition[SIf.Cur.iActualDistributionIndex]];
					me.StateMachine.intStateNext := PTS_CmdState.cSTA_WaitPaper;
				END_IF
			ELSE
				IF ((NOT SIf.Cfg.bolEntrySensorAvailable) OR (SIf.In.bolPaperAtBeltExit.intern)) THEN
//					SIf.Cur.rInOutPosition := SIf.Cfg.aFixPosDef[SIf.Par.eMode];
					me.StateMachine.intStateNext := PTS_CmdState.cSTA_WaitPaper;
				END_IF
		END_CASE

		CASE me.intCmd OF
			BASE_PLC.cCMD_STOP:
				me.StateMachine.intStateNext := BASE_PLC.cSTA_STOPBusy;
			PTS_CmdState.cCMD_STANDBY:
				me.StateMachine.intStateNext := PTS_CmdState.cSTA_STANDBYBusy;
		END_CASE
	END_IF


//--------------------------------------------------------------------------------------
// Exit action
	IF (me.StateMachine.intState<>me.StateMachine.intStateNext) THEN
		;
	END_IF
END_METHOD

{attribute 'object_name' := 'sta_RUNBusy'}
METHOD PROTECTED sta_RUNBusy : BOOL
// state implemetation
//--------------------------------------------------------------------------------------
// Entry action
IF (me.StateMachine.intState<>me.StateMachine.intStateLastCycle) THEN
	me.StateMachine.intStateLastCycle := me.StateMachine.intState;

	CASE SIf.Par.eMode OF
		E_PTS_MODE.Automatic:
			pfbAlarmCtrl^.setAlarm(CIf.Info.intCtrlId,INT_TO_UINT(E_ALM_PTS.ModeParameter),0,ADR(SIf.Alm),E_AlmState.RST,CIf.Job.eMe_ActivAlmClass);
(*
			IF SIf.Cfg.bolBarcodeReaderAvailable (* AND BCR has a new barcode read *) THEN
				me.StateMachine.intStateNext := PTS_CmdState.cSTA_GetItemBusy;
			ELSE
				pfbAlarmCtrl^.setAlarm(CIf.Info.intCtrlId,INT_TO_UINT(E_ALM_PTS.ModeParameter),0,ADR(SIf.Alm),E_AlmState.RST,CIf.Job.eMe_ActivAlmClass);
			END_IF
*)
		E_PTS_MODE.Distribute:
			SIf.Cur.rInOutPosition := SIf.Cfg.aFixPosDef[SIf.Cfg.aDistributionPositionDefinition[SIf.Cur.iActualDistributionIndex]];

		ELSE
			SIf.Cur.rInOutPosition := SIf.Cfg.aFixPosDef[SIf.Par.eMode];
	END_CASE

	(*p_fbMalteser^.CtrlSIf^.Par.*)intTurnDirection := E_TURN_DIRECTION.AUTOMATIC;
	(*p_fbMalteser^.CtrlSIf^.Par.*)uinPositionToGo := SIf.Cur.rInOutPosition.uinOutput;

	IF (SIf.Cfg.bolRaxEnable = FALSE) THEN
		IF SIf.Cfg.bolPositionMalteserEnable THEN
			p_fbMalteser^.CtrlCIf^.Job.intACmd := MDC_CmdState.cCMD_PREPOSITION;
	
			me.SubStateMachine.intState := PTS_CmdState.cSUB_PREPOSITIONbusy;
			me.SubStateMachine.intStateNext := PTS_CmdState.cSUB_PREPOSITIONbusy;
		ELSE	
			p_fbMalteser^.CtrlCIf^.Job.intACmd := BASE_PLC.cCMD_RUN;
	
			me.SubStateMachine.intState := PTS_CmdState.cSUB_WAIT_DONE;
			me.SubStateMachine.intStateNext := PTS_CmdState.cSUB_WAIT_DONE;
		END_IF
	END_IF
	
	p_fbBelt^.CtrlSIf^.Par.intDirection := E_BELT_DIRECTION.FORWARD;
	pBeltCIf^.Job.intACmd := BASE_PLC.cCMD_RUN;
END_IF


//--------------------------------------------------------------------------------------
// Cyclic action
IF (me.StateMachine.intState=me.StateMachine.intStateLastCycle) THEN

	IF (SIf.Cfg.bolRaxEnable) THEN
		me.StateMachine.intStateNext := cSTA_RUN;
	ELSE
		//--------------------------------------------------------------------------------------
		// sub state machine for sequence
		CASE me.SubStateMachine.intState OF
			//--------------------------------------------------------------------------------------
			PTS_CmdState.cSUB_PREPOSITIONbusy:
				IF (p_fbMalteser^.CtrlCIf^.Job.intState = MDC_CmdState.cSTA_PREPOSITION) THEN
					p_fbMalteser^.CtrlCIf^.Job.intACmd := BASE_PLC.cCMD_RUN;
					me.SubStateMachine.intStateNext := PTS_CmdState.cSUB_WAIT_DONE;
				END_IF
			//--------------------------------------------------------------------------------------
			PTS_CmdState.cSUB_WAIT_DONE:
				IF (p_fbMalteser^.CtrlCIf^.Job.intState = MDC_CmdState.cSTA_InPosition) 
				  AND (pBeltCIf^.Job.intState = BASE_PLC.cSTA_RUN) THEN
		//			SIf.Cur.udiPaperInTurnDelayTime := 150000 / p_fbBelt^.CtrlSIf^.Par.uinBeltSpeed;
		//			SIf.Cur.udiPaperOutTurnDelayTime := CalculateOutputDelay(p_fbBelt^.CtrlSIf^.Par.uinBeltSpeed,SIf.Cur.udiPaperInTurnDelayTime);
					me.StateMachine.intStateNext := BASE_PLC.cSTA_RUN;
				END_IF
			//--------------------------------------------------------------------------------------
		END_CASE
	END_IF
	
	IF SIf.In.bolPaperAvailable.intern THEN
		me.StateMachine.intStateNext := PTS_CmdState.cSTA_WaitPaper;
	END_IF
END_IF


//--------------------------------------------------------------------------------------
// Exit action
IF (me.StateMachine.intState<>me.StateMachine.intStateNext) THEN
	;
END_IF
END_METHOD

{attribute 'object_name' := 'sta_STANDBY'}
METHOD PROTECTED sta_STANDBY : BOOL
// state implemetation
//--------------------------------------------------------------------------------------
// Entry action
	IF (me.StateMachine.intState<>me.StateMachine.intStateLastCycle) THEN
		me.StateMachine.intStateLastCycle := me.StateMachine.intState;
		CIf.Job.intACmd := BASE_PLC.cCMD_DONE;
		CIf.Job.intMCmd := BASE_PLC.cCMD_DONE;
	END_IF


//--------------------------------------------------------------------------------------
// Cyclic action
	IF (me.StateMachine.intState = me.StateMachine.intStateLastCycle) THEN
		CASE me.intCmd OF
			BASE_PLC.cCMD_RUN:
				me.StateMachine.intStateNext := BASE_PLC.cSTA_RUNBusy;
			BASE_PLC.cCMD_STOP:
				me.StateMachine.intStateNext := BASE_PLC.cSTA_STOPBusy;
		END_CASE
	END_IF


//--------------------------------------------------------------------------------------
// Exit action
	IF (me.StateMachine.intState<>me.StateMachine.intStateNext) THEN
		;
	END_IF
END_METHOD

{attribute 'object_name' := 'sta_STANDBYBusy'}
METHOD PROTECTED sta_STANDBYBusy : BOOL
// state implemetation
//--------------------------------------------------------------------------------------
// Entry action
	IF (me.StateMachine.intState<>me.StateMachine.intStateLastCycle) THEN
		me.StateMachine.intStateLastCycle := me.StateMachine.intState;
		
		CASE SIf.Par.eMode OF
			E_PTS_MODE.Automatic:
				uinPositionToGo := SIf.Cfg.aDefaultAutoPos;
			E_PTS_MODE.Distribute:
				uinPositionToGo := SIf.Cfg.aFixPosDef[SIf.Cfg.aDistributionPositionDefinition[SIf.Cur.iActualDistributionIndex]].uinInput;
			ELSE
				uinPositionToGo := SIf.Cfg.aFixPosDef[SIf.Par.eMode].uinInput;
		END_CASE

		// p_fbMalteser^.SetPositionToGo(uinPositionToGo);

		IF (SIf.Cfg.bolRaxEnable) THEN
			IF p_fbRAX^.CtrlSIf^.Cur.dinPosition_0_1Deg <> uinPositionToGo*90*10 THEN
				pRaxCIf^.Job.intACmd := RAX_CmdState.cCMD_TURN;
			END_IF
		ELSE
			IF p_fbMalteser^.ActualPosition <> uinPositionToGo THEN
				pMalteserCIf^.Job.intACmd := MDC_CmdState.cCMD_TURN;
			END_IF
		END_IF
		
		pBeltCIf^.Job.intACmd := BASE_PLC.cCMD_STOP;
		
		me.SubStateMachine.intState 	:= PTS_CmdState.cSUB_TURNbusy;
		me.SubStateMachine.intStateNext := PTS_CmdState.cSUB_TURNbusy;
	END_IF


//--------------------------------------------------------------------------------------
// Cyclic action
	IF (me.StateMachine.intState=me.StateMachine.intStateLastCycle) THEN
		IF (SIf.Cfg.bolRaxEnable) THEN
			CASE me.SubStateMachine.intState OF
				PTS_CmdState.cSUB_TURNbusy:
					IF    (p_fbRAX^.CtrlSIf^.Cur.dinPosition_0_1Deg = p_fbRAX^.CtrlSIf^.Par.dinPos_0_1Deg) 
					  AND (  (pRaxCIf^.Job.intState = cSTA_STOP) 
						   OR(pRaxCIf^.Job.intState = cSTA_TURN))THEN 
						pRaxCIf^.Job.intACmd := BASE_PLC.cCMD_RUN;
						me.SubStateMachine.intStateNext := PTS_CmdState.cSUB_TURNDONE;
					END_IF
				PTS_CmdState.cSUB_TURNDONE:
					IF (pRaxCIf^.Job.intState = cSTA_STOP) 
					  AND ((pBeltCIf^.Job.intState = BASE_PLC.cSTA_OFF) OR (pBeltCIf^.Job.intState = BASE_PLC.cSTA_STOP)) THEN
						me.StateMachine.intStateNext := PTS_CmdState.cSTA_STANDBY;
					END_IF
			END_CASE
		ELSE
			CASE me.SubStateMachine.intState OF
				PTS_CmdState.cSUB_TURNbusy:
					IF    (p_fbMalteser^.CtrlSIf^.Cur.uintActualPosition = p_fbMalteser^.CtrlSIf^.Par.uinPositionToGo) 
					  AND (  (pMalteserCIf^.Job.intState = MDC_CmdState.cSTA_InPosition) 
						   OR(pMalteserCIf^.Job.intState = MDC_CmdState.cSTA_TURNDONE))THEN 
						pMalteserCIf^.Job.intACmd := BASE_PLC.cCMD_RUN;
						me.SubStateMachine.intStateNext := PTS_CmdState.cSUB_TURNDONE;
					END_IF
				PTS_CmdState.cSUB_TURNDONE:
					IF (pMalteserCIf^.Job.intState = MDC_CmdState.cSTA_InPosition) 
					  AND ((pBeltCIf^.Job.intState = BASE_PLC.cSTA_OFF) OR (pBeltCIf^.Job.intState = BASE_PLC.cSTA_STOP)) THEN
						me.StateMachine.intStateNext := PTS_CmdState.cSTA_STANDBY;
					END_IF
			END_CASE	
		END_IF
	END_IF


